Yaskawa INFORM job: DEMO_ROOF_UPPER_0625_3PAINT_38.JBI

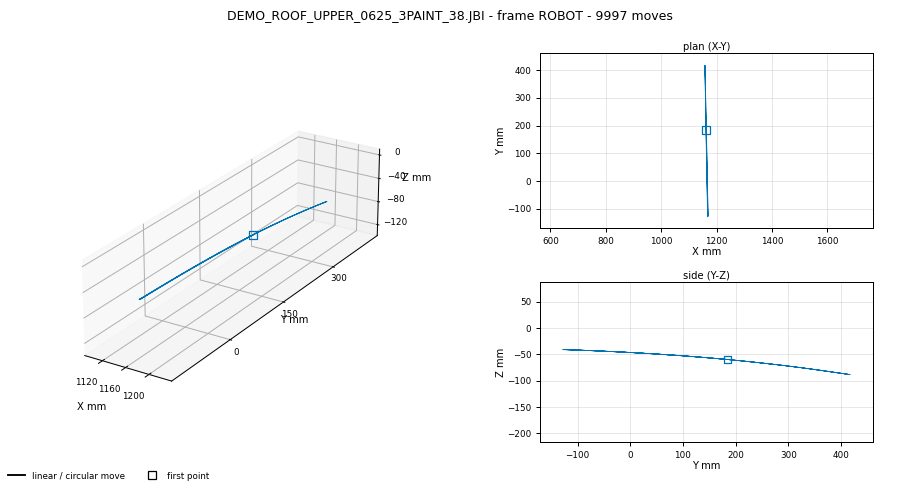
[picture p0: tool path of DEMO_ROOF_UPPER_0625_3PAINT_38.JBI in frame ROBOT, 9997 of 9997 moves have a stored position in this frame; points joined in program order, loops and branches not executed]
/JOB
//NAME DEMO_ROOF_UPPER_0625_3PAINT38
//POS
///NPOS 9997,0,0,0,0,0
///TOOL 0
///USER 0
///POSTYPE ROBOT
///RECTAN
///RCONF 1,0,0,0,0,0,0,0,0,0,0,0,0,0,0,0,0,0,0,0,0,0,0,0
C00000=1163.318,184.615,-59.683,-178.143,6.943,148.746
C00001=1163.323,184.345,-59.658,-178.145,6.942,148.747
C00002=1163.328,184.076,-59.633,-178.149,6.939,148.747
C00003=1163.333,183.807,-59.608,-178.152,6.936,148.747
C00004=1163.338,183.537,-59.582,-178.155,6.935,148.748
C00005=1163.342,183.288,-59.560,-178.157,6.933,148.748
C00006=1163.347,183.038,-59.537,-178.160,6.930,148.748
C00007=1163.352,182.789,-59.514,-178.163,6.928,148.748
C00008=1163.357,182.541,-59.491,-178.166,6.926,148.749
C00009=1163.361,182.292,-59.468,-178.169,6.924,148.749
C00010=1163.366,182.043,-59.445,-178.171,6.922,148.749
C00011=1163.370,181.794,-59.423,-178.174,6.920,148.750
C00012=1163.375,181.545,-59.399,-178.176,6.918,148.750
C00013=1163.379,181.297,-59.377,-178.180,6.916,148.750
C00014=1163.384,181.048,-59.353,-178.182,6.914,148.750
C00015=1163.389,180.799,-59.330,-178.185,6.912,148.751
C00016=1163.393,180.549,-59.308,-178.188,6.909,148.751
C00017=1163.398,180.300,-59.285,-178.190,6.907,148.752
C00018=1163.402,180.052,-59.262,-178.193,6.905,148.752
C00019=1163.407,179.803,-59.240,-178.195,6.904,148.752
C00020=1163.411,179.554,-59.217,-178.199,6.901,148.752
C00021=1163.416,179.305,-59.193,-178.201,6.899,148.753
C00022=1163.422,179.056,-59.171,-178.204,6.898,148.753
C00023=1163.426,178.807,-59.148,-178.206,6.895,148.753
C00024=1163.430,178.558,-59.125,-178.209,6.893,148.754
C00025=1163.435,178.309,-59.103,-178.212,6.891,148.754
C00026=1163.440,178.061,-59.080,-178.215,6.889,148.754
C00027=1163.444,177.811,-59.058,-178.217,6.887,148.754
C00028=1163.449,177.562,-59.035,-178.220,6.885,148.755
C00029=1163.453,177.314,-59.012,-178.223,6.883,148.755
C00030=1163.458,177.065,-58.990,-178.226,6.881,148.755
C00031=1163.462,176.816,-58.967,-178.228,6.879,148.756
C00032=1163.468,176.567,-58.945,-178.231,6.876,148.756
C00033=1163.472,176.318,-58.922,-178.234,6.875,148.756
C00034=1163.477,176.069,-58.899,-178.237,6.873,148.757
C00035=1163.482,175.821,-58.877,-178.239,6.871,148.757
C00036=1163.486,175.571,-58.855,-178.242,6.869,148.757
C00037=1163.491,175.322,-58.831,-178.245,6.867,148.758
C00038=1163.495,175.074,-58.810,-178.247,6.865,148.758
C00039=1163.500,174.824,-58.786,-178.250,6.863,148.758
C00040=1163.504,174.575,-58.764,-178.253,6.861,148.759
C00041=1163.510,174.327,-58.741,-178.256,6.859,148.759
C00042=1163.514,174.077,-58.719,-178.258,6.857,148.759
C00043=1163.518,173.829,-58.696,-178.261,6.855,148.760
C00044=1163.523,173.580,-58.674,-178.264,6.853,148.760
C00045=1163.528,173.330,-58.652,-178.267,6.851,148.760
C00046=1163.532,173.082,-58.629,-178.270,6.849,148.761
C00047=1163.537,172.833,-58.607,-178.272,6.847,148.761
C00048=1163.542,172.583,-58.585,-178.274,6.845,148.761
C00049=1163.547,172.335,-58.562,-178.277,6.843,148.761
C00050=1163.551,172.086,-58.540,-178.280,6.841,148.762
C00051=1163.555,171.836,-58.518,-178.283,6.839,148.762
C00052=1163.560,171.588,-58.496,-178.286,6.837,148.763
C00053=1163.565,171.339,-58.473,-178.289,6.835,148.763
C00054=1163.570,171.090,-58.451,-178.291,6.833,148.763
C00055=1163.574,170.841,-58.428,-178.294,6.831,148.763
C00056=1163.579,170.592,-58.406,-178.297,6.829,148.764
C00057=1163.584,170.343,-58.384,-178.299,6.827,148.764
C00058=1163.588,170.094,-58.362,-178.302,6.825,148.765
C00059=1163.593,169.845,-58.339,-178.305,6.824,148.765
C00060=1163.598,169.596,-58.317,-178.308,6.821,148.765
C00061=1163.602,169.347,-58.295,-178.310,6.819,148.765
C00062=1163.607,169.098,-58.273,-178.313,6.817,148.766
C00063=1163.612,168.849,-58.251,-178.316,6.815,148.766
C00064=1163.616,168.600,-58.228,-178.318,6.814,148.766
C00065=1163.621,168.352,-58.207,-178.322,6.811,148.767
C00066=1163.625,168.102,-58.185,-178.324,6.809,148.767
C00067=1163.630,167.854,-58.163,-178.326,6.807,148.767
C00068=1163.635,167.604,-58.140,-178.329,6.806,148.768
C00069=1163.640,167.356,-58.119,-178.332,6.804,148.768
C00070=1163.644,167.106,-58.096,-178.335,6.802,148.768
C00071=1163.649,166.858,-58.075,-178.338,6.800,148.769
C00072=1163.654,166.608,-58.053,-178.341,6.798,148.769
C00073=1163.658,166.360,-58.030,-178.343,6.796,148.770
C00074=1163.663,166.111,-58.008,-178.346,6.794,148.770
C00075=1163.668,165.862,-57.986,-178.348,6.792,148.770
C00076=1163.672,165.613,-57.964,-178.351,6.790,148.770
C00077=1163.677,165.364,-57.942,-178.354,6.788,148.771
C00078=1163.681,165.115,-57.920,-178.357,6.786,148.771
C00079=1163.686,164.866,-57.899,-178.359,6.784,148.772
C00080=1163.691,164.617,-57.877,-178.362,6.783,148.772
C00081=1163.695,164.368,-57.855,-178.365,6.781,148.772
C00082=1163.700,164.119,-57.833,-178.368,6.779,148.773
C00083=1163.705,163.870,-57.811,-178.370,6.777,148.773
C00084=1163.710,163.621,-57.789,-178.373,6.774,148.773
C00085=1163.715,163.371,-57.767,-178.376,6.773,148.774
C00086=1163.720,163.122,-57.746,-178.378,6.771,148.774
C00087=1163.724,162.873,-57.724,-178.381,6.769,148.774
C00088=1163.729,162.624,-57.702,-178.384,6.767,148.775
C00089=1163.734,162.376,-57.680,-178.386,6.766,148.775
C00090=1163.738,162.126,-57.658,-178.389,6.764,148.775
C00091=1163.743,161.878,-57.637,-178.392,6.761,148.776
C00092=1163.747,161.628,-57.615,-178.395,6.760,148.776
C00093=1163.752,161.379,-57.594,-178.397,6.758,148.776
C00094=1163.757,161.131,-57.572,-178.400,6.756,148.777
C00095=1163.761,160.881,-57.550,-178.403,6.754,148.777
C00096=1163.766,160.633,-57.528,-178.405,6.752,148.777
C00097=1163.770,160.383,-57.506,-178.408,6.751,148.778
C00098=1163.775,160.135,-57.485,-178.411,6.749,148.778
C00099=1163.780,159.885,-57.464,-178.414,6.746,148.778
C00100=1163.785,159.636,-57.441,-178.417,6.745,148.779
C00101=1163.790,159.387,-57.420,-178.419,6.743,148.779
C00102=1163.794,159.139,-57.399,-178.422,6.741,148.780
C00103=1163.798,158.889,-57.377,-178.425,6.739,148.780
C00104=1163.803,158.640,-57.356,-178.428,6.738,148.780
C00105=1163.809,158.371,-57.332,-178.430,6.736,148.781
C00106=1163.813,158.103,-57.309,-178.434,6.733,148.781
C00107=1163.819,157.833,-57.286,-178.436,6.731,148.781
C00108=1163.823,157.564,-57.263,-178.440,6.729,148.782
C00109=1163.828,157.316,-57.241,-178.442,6.727,148.782
C00110=1163.833,157.066,-57.220,-178.445,6.725,148.783
C00111=1163.838,156.817,-57.198,-178.448,6.724,148.783
C00112=1163.843,156.568,-57.176,-178.450,6.722,148.783
C00113=1163.848,156.319,-57.155,-178.453,6.720,148.784
C00114=1163.852,156.071,-57.134,-178.456,6.718,148.784
C00115=1163.856,155.821,-57.113,-178.458,6.717,148.784
C00116=1163.861,155.572,-57.091,-178.461,6.715,148.785
C00117=1163.866,155.324,-57.070,-178.464,6.713,148.785
C00118=1163.871,155.074,-57.048,-178.466,6.711,148.785
C00119=1163.876,154.825,-57.027,-178.469,6.709,148.786
C00120=1163.880,154.576,-57.006,-178.472,6.707,148.786
C00121=1163.885,154.327,-56.985,-178.475,6.705,148.786
C00122=1163.889,154.077,-56.963,-178.477,6.703,148.787
C00123=1163.894,153.829,-56.942,-178.480,6.702,148.787
C00124=1163.899,153.580,-56.921,-178.483,6.700,148.788
C00125=1163.904,153.331,-56.899,-178.485,6.698,148.788
C00126=1163.909,153.082,-56.879,-178.488,6.696,148.788
C00127=1163.913,152.833,-56.856,-178.491,6.695,148.789
C00128=1163.918,152.584,-56.836,-178.494,6.693,148.789
C00129=1163.923,152.334,-56.815,-178.496,6.691,148.790
C00130=1163.928,152.086,-56.793,-178.499,6.689,148.790
C00131=1163.932,151.836,-56.772,-178.502,6.688,148.790
C00132=1163.936,151.587,-56.751,-178.504,6.686,148.791
C00133=1163.941,151.338,-56.730,-178.507,6.684,148.791
C00134=1163.947,151.089,-56.709,-178.510,6.682,148.791
C00135=1163.951,150.841,-56.688,-178.513,6.680,148.792
C00136=1163.956,150.591,-56.667,-178.516,6.678,148.792
C00137=1163.960,150.341,-56.646,-178.518,6.676,148.793
C00138=1163.965,150.093,-56.625,-178.521,6.675,148.793
C00139=1163.970,149.844,-56.604,-178.524,6.673,148.793
C00140=1163.975,149.594,-56.583,-178.527,6.671,148.794
C00141=1163.979,149.346,-56.562,-178.529,6.669,148.794
C00142=1163.984,149.097,-56.541,-178.532,6.668,148.794
C00143=1163.989,148.848,-56.520,-178.535,6.666,148.795
C00144=1163.993,148.598,-56.499,-178.537,6.664,148.795
C00145=1163.998,148.349,-56.477,-178.540,6.663,148.796
C00146=1164.003,148.100,-56.457,-178.543,6.661,148.796
C00147=1164.008,147.851,-56.436,-178.545,6.659,148.796
C00148=1164.013,147.602,-56.415,-178.548,6.657,148.797
C00149=1164.017,147.354,-56.394,-178.551,6.656,148.797
C00150=1164.022,147.104,-56.373,-178.554,6.654,148.798
C00151=1164.027,146.855,-56.353,-178.556,6.652,148.798
C00152=1164.031,146.605,-56.331,-178.559,6.650,148.798
C00153=1164.036,146.356,-56.311,-178.562,6.649,148.799
C00154=1164.041,146.107,-56.290,-178.564,6.647,148.799
C00155=1164.045,145.859,-56.269,-178.567,6.645,148.799
C00156=1164.050,145.610,-56.248,-178.570,6.643,148.800
C00157=1164.055,145.361,-56.227,-178.572,6.642,148.800
C00158=1164.060,145.111,-56.206,-178.575,6.640,148.801
C00159=1164.064,144.862,-56.186,-178.578,6.638,148.801
C00160=1164.069,144.613,-56.165,-178.581,6.636,148.801
C00161=1164.074,144.364,-56.145,-178.583,6.635,148.802
C00162=1164.079,144.115,-56.124,-178.586,6.633,148.802
C00163=1164.083,143.866,-56.103,-178.589,6.631,148.803
C00164=1164.089,143.617,-56.082,-178.591,6.630,148.803
C00165=1164.093,143.368,-56.062,-178.594,6.628,148.803
C00166=1164.098,143.118,-56.041,-178.597,6.626,148.804
C00167=1164.102,142.869,-56.020,-178.600,6.625,148.804
C00168=1164.107,142.620,-56.000,-178.603,6.623,148.805
C00169=1164.112,142.371,-55.979,-178.605,6.621,148.805
C00170=1164.116,142.122,-55.959,-178.608,6.619,148.805
C00171=1164.121,141.872,-55.938,-178.611,6.618,148.806
C00172=1164.126,141.624,-55.917,-178.613,6.616,148.806
C00173=1164.130,141.375,-55.897,-178.616,6.614,148.807
C00174=1164.135,141.125,-55.876,-178.619,6.613,148.807
C00175=1164.140,140.876,-55.856,-178.622,6.611,148.807
C00176=1164.145,140.627,-55.835,-178.624,6.609,148.808
C00177=1164.149,140.378,-55.814,-178.627,6.607,148.808
C00178=1164.154,140.129,-55.794,-178.630,6.606,148.809
C00179=1164.159,139.880,-55.773,-178.632,6.604,148.809
C00180=1164.164,139.630,-55.753,-178.635,6.602,148.809
C00181=1164.169,139.382,-55.733,-178.638,6.600,148.810
C00182=1164.174,139.133,-55.712,-178.640,6.599,148.810
C00183=1164.178,138.884,-55.692,-178.643,6.597,148.810
C00184=1164.183,138.635,-55.672,-178.646,6.596,148.811
C00185=1164.188,138.386,-55.651,-178.649,6.594,148.811
C00186=1164.193,138.136,-55.631,-178.652,6.592,148.812
C00187=1164.197,137.887,-55.611,-178.654,6.590,148.812
C00188=1164.202,137.638,-55.590,-178.657,6.589,148.813
C00189=1164.207,137.389,-55.569,-178.660,6.587,148.813
C00190=1164.212,137.139,-55.550,-178.663,6.585,148.813
C00191=1164.216,136.890,-55.529,-178.665,6.583,148.814
C00192=1164.220,136.642,-55.509,-178.668,6.582,148.814
C00193=1164.226,136.392,-55.488,-178.671,6.580,148.815
C00194=1164.230,136.143,-55.468,-178.673,6.579,148.815
C00195=1164.235,135.894,-55.448,-178.676,6.577,148.815
C00196=1164.240,135.646,-55.428,-178.679,6.576,148.816
C00197=1164.245,135.396,-55.408,-178.681,6.574,148.816
C00198=1164.250,135.147,-55.387,-178.684,6.572,148.817
C00199=1164.254,134.898,-55.367,-178.687,6.571,148.817
C00200=1164.259,134.648,-55.347,-178.690,6.569,148.818
C00201=1164.263,134.399,-55.327,-178.692,6.567,148.818
C00202=1164.269,134.150,-55.306,-178.695,6.566,148.818
C00203=1164.274,133.901,-55.287,-178.698,6.564,148.819
C00204=1164.278,133.652,-55.266,-178.700,6.562,148.819
C00205=1164.283,133.403,-55.247,-178.703,6.560,148.820
C00206=1164.287,133.154,-55.226,-178.706,6.559,148.820
C00207=1164.292,132.905,-55.206,-178.709,6.557,148.821
C00208=1164.297,132.655,-55.186,-178.712,6.556,148.821
C00209=1164.302,132.386,-55.164,-178.714,6.554,148.821
C00210=1164.307,132.118,-55.143,-178.717,6.552,148.822
C00211=1164.313,131.849,-55.121,-178.720,6.551,148.822
C00212=1164.318,131.580,-55.100,-178.723,6.549,148.823
C00213=1164.323,131.332,-55.080,-178.726,6.547,148.823
C00214=1164.327,131.083,-55.060,-178.728,6.546,148.823
C00215=1164.332,130.833,-55.039,-178.731,6.544,148.824
C00216=1164.337,130.584,-55.020,-178.734,6.542,148.824
C00217=1164.342,130.335,-54.999,-178.737,6.540,148.825
C00218=1164.347,130.086,-54.980,-178.740,6.539,148.825
C00219=1164.351,129.837,-54.960,-178.742,6.538,148.826
C00220=1164.356,129.588,-54.940,-178.745,6.536,148.826
C00221=1164.361,129.339,-54.920,-178.747,6.535,148.826
C00222=1164.366,129.090,-54.900,-178.750,6.533,148.827
C00223=1164.371,128.840,-54.881,-178.753,6.531,148.827
C00224=1164.375,128.591,-54.860,-178.755,6.529,148.828
C00225=1164.380,128.342,-54.841,-178.758,6.528,148.828
C00226=1164.385,128.093,-54.821,-178.761,6.526,148.829
C00227=1164.390,127.844,-54.801,-178.764,6.525,148.829
C00228=1164.394,127.594,-54.781,-178.766,6.524,148.829
C00229=1164.399,127.345,-54.762,-178.769,6.522,148.830
C00230=1164.404,127.096,-54.742,-178.772,6.520,148.830
C00231=1164.409,126.847,-54.722,-178.774,6.519,148.831
C00232=1164.414,126.597,-54.702,-178.777,6.517,148.831
C00233=1164.418,126.348,-54.682,-178.780,6.515,148.832
C00234=1164.423,126.099,-54.663,-178.783,6.514,148.832
C00235=1164.428,125.850,-54.643,-178.786,6.512,148.832
C00236=1164.432,125.601,-54.624,-178.788,6.510,148.833
C00237=1164.437,125.352,-54.604,-178.790,6.509,148.833
C00238=1164.442,125.103,-54.584,-178.793,6.508,148.834
C00239=1164.447,124.853,-54.565,-178.796,6.506,148.834
C00240=1164.452,124.604,-54.545,-178.799,6.505,148.835
C00241=1164.456,124.355,-54.525,-178.802,6.503,148.835
C00242=1164.461,124.106,-54.505,-178.804,6.501,148.835
C00243=1164.467,123.857,-54.486,-178.807,6.499,148.836
C00244=1164.471,123.607,-54.466,-178.809,6.498,148.836
C00245=1164.475,123.358,-54.447,-178.812,6.497,148.837
C00246=1164.481,123.109,-54.428,-178.815,6.495,148.837
C00247=1164.485,122.860,-54.408,-178.818,6.494,148.838
C00248=1164.490,122.611,-54.388,-178.821,6.492,148.838
C00249=1164.495,122.362,-54.369,-178.823,6.490,148.838
C00250=1164.500,122.112,-54.349,-178.826,6.489,148.839
C00251=1164.504,121.863,-54.330,-178.829,6.488,148.840
C00252=1164.509,121.614,-54.311,-178.831,6.486,148.840
C00253=1164.514,121.365,-54.291,-178.834,6.485,148.840
C00254=1164.519,121.116,-54.272,-178.837,6.483,148.841
C00255=1164.524,120.866,-54.252,-178.839,6.481,148.841
C00256=1164.528,120.617,-54.233,-178.842,6.479,148.842
C00257=1164.533,120.368,-54.214,-178.845,6.479,148.842
C00258=1164.538,120.119,-54.194,-178.847,6.477,148.843
C00259=1164.544,119.870,-54.175,-178.850,6.475,148.843
C00260=1164.548,119.620,-54.156,-178.853,6.474,148.843
C00261=1164.552,119.371,-54.136,-178.856,6.472,148.844
C00262=1164.558,119.122,-54.117,-178.859,6.471,148.844
C00263=1164.562,118.872,-54.097,-178.861,6.470,148.845
C00264=1164.567,118.624,-54.078,-178.864,6.468,148.845
C00265=1164.572,118.374,-54.059,-178.866,6.466,148.846
C00266=1164.577,118.125,-54.039,-178.869,6.464,148.846
C00267=1164.581,117.876,-54.020,-178.872,6.463,148.847
C00268=1164.586,117.627,-54.001,-178.874,6.462,148.847
C00269=1164.591,117.378,-53.981,-178.877,6.461,148.847
C00270=1164.595,117.128,-53.962,-178.880,6.459,148.848
C00271=1164.601,116.880,-53.943,-178.883,6.457,148.848
C00272=1164.606,116.629,-53.924,-178.886,6.456,148.849
C00273=1164.610,116.381,-53.905,-178.888,6.455,148.849
C00274=1164.615,116.131,-53.886,-178.891,6.453,148.850
C00275=1164.620,115.882,-53.866,-178.893,6.451,148.850
C00276=1164.624,115.633,-53.847,-178.896,6.450,148.850
C00277=1164.630,115.384,-53.828,-178.899,6.448,148.851
C00278=1164.635,115.134,-53.809,-178.901,6.447,148.852
C00279=1164.639,114.886,-53.790,-178.904,6.446,148.852
C00280=1164.644,114.636,-53.771,-178.907,6.444,148.852
C00281=1164.649,114.387,-53.752,-178.910,6.443,148.853
C00282=1164.654,114.137,-53.733,-178.913,6.441,148.853
C00283=1164.659,113.888,-53.714,-178.915,6.440,148.854
C00284=1164.663,113.639,-53.695,-178.918,6.438,148.854
C00285=1164.668,113.390,-53.676,-178.920,6.437,148.855
C00286=1164.673,113.140,-53.657,-178.923,6.435,148.855
C00287=1164.678,112.891,-53.638,-178.926,6.433,148.856
C00288=1164.682,112.642,-53.619,-178.928,6.433,148.856
C00289=1164.688,112.393,-53.600,-178.931,6.431,148.856
C00290=1164.693,112.144,-53.581,-178.934,6.430,148.857
C00291=1164.697,111.895,-53.562,-178.937,6.428,148.857
C00292=1164.703,111.645,-53.543,-178.939,6.427,148.858
C00293=1164.707,111.396,-53.524,-178.942,6.425,148.858
C00294=1164.712,111.147,-53.505,-178.945,6.424,148.859
C00295=1164.716,110.897,-53.487,-178.948,6.422,148.859
C00296=1164.722,110.648,-53.467,-178.950,6.420,148.860
C00297=1164.726,110.400,-53.449,-178.953,6.419,148.860
C00298=1164.731,110.150,-53.430,-178.955,6.418,148.861
C00299=1164.736,109.901,-53.411,-178.958,6.416,148.861
C00300=1164.741,109.651,-53.392,-178.961,6.415,148.862
C00301=1164.746,109.402,-53.373,-178.963,6.414,148.862
C00302=1164.750,109.153,-53.355,-178.966,6.412,148.862
C00303=1164.755,108.903,-53.336,-178.969,6.411,148.863
C00304=1164.760,108.655,-53.317,-178.972,6.409,148.863
C00305=1164.765,108.405,-53.298,-178.974,6.408,148.864
C00306=1164.770,108.156,-53.279,-178.977,6.406,148.864
C00307=1164.775,107.907,-53.261,-178.980,6.405,148.865
C00308=1164.779,107.657,-53.242,-178.983,6.403,148.865
C00309=1164.784,107.408,-53.224,-178.985,6.402,148.866
C00310=1164.789,107.159,-53.204,-178.988,6.401,148.866
C00311=1164.794,106.910,-53.186,-178.991,6.399,148.867
C00312=1164.799,106.660,-53.168,-178.993,6.398,148.867
C00313=1164.804,106.392,-53.147,-178.996,6.397,148.868
C00314=1164.809,106.123,-53.127,-178.999,6.395,148.868
C00315=1164.814,105.855,-53.108,-179.002,6.394,148.869
C00316=1164.820,105.587,-53.087,-179.005,6.392,148.869
C00317=1164.825,105.338,-53.069,-179.007,6.391,148.870
C00318=1164.829,105.089,-53.050,-179.010,6.389,148.870
C00319=1164.835,104.839,-53.031,-179.013,6.388,148.871
C00320=1164.839,104.590,-53.013,-179.016,6.387,148.871
C00321=1164.843,104.341,-52.994,-179.018,6.385,148.872
C00322=1164.848,104.091,-52.976,-179.021,6.383,148.872
C00323=1164.854,103.842,-52.958,-179.024,6.383,148.873
C00324=1164.858,103.593,-52.939,-179.026,6.381,148.873
C00325=1164.863,103.343,-52.921,-179.029,6.379,148.873
C00326=1164.869,103.094,-52.902,-179.032,6.378,148.874
C00327=1164.873,102.845,-52.883,-179.034,6.377,148.874
C00328=1164.877,102.596,-52.865,-179.037,6.375,148.875
C00329=1164.882,102.346,-52.847,-179.040,6.374,148.875
C00330=1164.888,102.097,-52.829,-179.042,6.373,148.876
C00331=1164.893,101.848,-52.810,-179.045,6.371,148.876
C00332=1164.897,101.598,-52.791,-179.048,6.370,148.877
C00333=1164.902,101.349,-52.774,-179.050,6.369,148.877
C00334=1164.908,101.100,-52.755,-179.053,6.367,148.878
C00335=1164.912,100.851,-52.737,-179.056,6.366,148.878
C00336=1164.916,100.601,-52.718,-179.059,6.364,148.879
C00337=1164.921,100.352,-52.700,-179.061,6.364,148.879
C00338=1164.926,100.103,-52.682,-179.064,6.362,148.880
C00339=1164.932,99.854,-52.663,-179.067,6.360,148.880
C00340=1164.936,99.604,-52.645,-179.069,6.360,148.881
C00341=1164.941,99.355,-52.626,-179.072,6.358,148.881
C00342=1164.946,99.106,-52.608,-179.075,6.356,148.882
C00343=1164.951,98.857,-52.590,-179.077,6.356,148.882
C00344=1164.956,98.608,-52.572,-179.080,6.354,148.883
C00345=1164.960,98.358,-52.554,-179.083,6.352,148.883
C00346=1164.966,98.108,-52.535,-179.085,6.351,148.883
C00347=1164.970,97.859,-52.517,-179.088,6.350,148.884
C00348=1164.975,97.610,-52.499,-179.091,6.348,148.885
C00349=1164.980,97.361,-52.482,-179.093,6.347,148.885
C00350=1164.985,97.112,-52.464,-179.096,6.346,148.886
C00351=1164.990,96.862,-52.445,-179.099,6.344,148.886
C00352=1164.994,96.612,-52.427,-179.101,6.343,148.886
C00353=1164.999,96.363,-52.409,-179.104,6.342,148.887
C00354=1165.004,96.114,-52.391,-179.107,6.340,148.887
C00355=1165.010,95.865,-52.373,-179.109,6.340,148.888
C00356=1165.015,95.615,-52.355,-179.112,6.338,148.889
C00357=1165.019,95.366,-52.336,-179.115,6.336,148.889
C00358=1165.024,95.116,-52.318,-179.117,6.336,148.889
C00359=1165.029,94.867,-52.300,-179.120,6.334,148.890
C00360=1165.034,94.618,-52.282,-179.123,6.333,148.890
C00361=1165.039,94.369,-52.264,-179.125,6.332,148.891
C00362=1165.044,94.120,-52.246,-179.129,6.330,148.892
C00363=1165.049,93.871,-52.228,-179.131,6.329,148.892
C00364=1165.053,93.621,-52.210,-179.133,6.328,148.892
C00365=1165.058,93.372,-52.193,-179.137,6.326,148.893
C00366=1165.063,93.122,-52.174,-179.139,6.325,148.893
C00367=1165.068,92.873,-52.156,-179.141,6.324,148.894
C00368=1165.073,92.624,-52.138,-179.145,6.322,148.894
C00369=1165.077,92.375,-52.120,-179.147,6.321,148.895
C00370=1165.083,92.125,-52.103,-179.150,6.320,148.895
C00371=1165.088,91.876,-52.085,-179.153,6.319,148.896
C00372=1165.092,91.627,-52.067,-179.155,6.318,148.896
C00373=1165.097,91.377,-52.049,-179.158,6.316,148.897
C00374=1165.102,91.128,-52.031,-179.161,6.315,148.897
C00375=1165.107,90.879,-52.014,-179.163,6.314,148.898
C00376=1165.112,90.630,-51.996,-179.166,6.312,148.898
C00377=1165.117,90.380,-51.978,-179.169,6.311,148.899
C00378=1165.122,90.131,-51.960,-179.171,6.310,148.899
C00379=1165.126,89.882,-51.942,-179.174,6.308,148.900
C00380=1165.132,89.632,-51.925,-179.176,6.308,148.900
C00381=1165.137,89.383,-51.907,-179.179,6.306,148.901
C00382=1165.141,89.133,-51.889,-179.182,6.304,148.901
C00383=1165.146,88.884,-51.871,-179.184,6.304,148.902
C00384=1165.151,88.634,-51.854,-179.187,6.302,148.902
C00385=1165.155,88.385,-51.836,-179.190,6.300,148.903
C00386=1165.160,88.136,-51.818,-179.193,6.300,148.903
C00387=1165.165,87.886,-51.801,-179.195,6.298,148.904
C00388=1165.170,87.637,-51.783,-179.197,6.297,148.904
C00389=1165.175,87.388,-51.765,-179.201,6.296,148.905
C00390=1165.180,87.138,-51.748,-179.203,6.294,148.905
C00391=1165.185,86.889,-51.730,-179.206,6.294,148.906
C00392=1165.189,86.640,-51.712,-179.209,6.292,148.906
C00393=1165.195,86.391,-51.696,-179.211,6.291,148.907
C00394=1165.200,86.142,-51.678,-179.214,6.290,148.907
C00395=1165.205,85.892,-51.660,-179.217,6.288,148.908
C00396=1165.210,85.643,-51.643,-179.219,6.287,148.908
C00397=1165.214,85.394,-51.625,-179.222,6.286,148.909
C00398=1165.220,85.144,-51.608,-179.224,6.285,148.909
C00399=1165.225,84.895,-51.590,-179.227,6.283,148.910
C00400=1165.229,84.646,-51.573,-179.230,6.283,148.910
C00401=1165.234,84.397,-51.555,-179.232,6.281,148.911
C00402=1165.239,84.147,-51.538,-179.236,6.280,148.912
C00403=1165.244,83.898,-51.520,-179.238,6.279,148.912
C00404=1165.249,83.648,-51.503,-179.240,6.277,148.912
C00405=1165.254,83.399,-51.485,-179.243,6.277,148.913
C00406=1165.259,83.149,-51.468,-179.246,6.275,148.913
C00407=1165.264,82.900,-51.450,-179.249,6.273,148.914
C00408=1165.268,82.650,-51.433,-179.251,6.273,148.915
C00409=1165.273,82.401,-51.415,-179.254,6.271,148.915
C00410=1165.279,82.152,-51.398,-179.256,6.270,148.916
C00411=1165.283,81.903,-51.381,-179.259,6.269,148.916
C00412=1165.288,81.653,-51.364,-179.261,6.268,148.916
C00413=1165.293,81.404,-51.346,-179.265,6.266,148.917
C00414=1165.298,81.155,-51.329,-179.267,6.265,148.918
C00415=1165.303,80.905,-51.312,-179.270,6.264,148.918
C00416=1165.308,80.656,-51.294,-179.273,6.263,148.919
C00417=1165.313,80.388,-51.276,-179.275,6.262,148.919
C00418=1165.318,80.119,-51.257,-179.278,6.260,148.920
C00419=1165.324,79.851,-51.238,-179.281,6.259,148.920
C00420=1165.329,79.583,-51.220,-179.284,6.257,148.921
C00421=1165.334,79.333,-51.203,-179.287,6.257,148.921
C00422=1165.339,79.083,-51.186,-179.289,6.255,148.922
C00423=1165.343,78.835,-51.168,-179.291,6.254,148.922
C00424=1165.349,78.585,-51.151,-179.295,6.253,148.923
C00425=1165.354,78.335,-51.134,-179.297,6.252,148.923
C00426=1165.359,78.087,-51.117,-179.300,6.251,148.924
C00427=1165.364,77.837,-51.099,-179.302,6.250,148.924
C00428=1165.368,77.588,-51.083,-179.305,6.248,148.925
C00429=1165.373,77.338,-51.065,-179.308,6.247,148.925
C00430=1165.378,77.089,-51.048,-179.310,6.246,148.926
C00431=1165.383,76.839,-51.031,-179.313,6.245,148.927
C00432=1165.388,76.590,-51.015,-179.316,6.244,148.927
C00433=1165.393,76.340,-50.997,-179.318,6.242,148.927
C00434=1165.397,76.092,-50.980,-179.321,6.242,148.928
C00435=1165.403,75.842,-50.963,-179.324,6.240,148.929
C00436=1165.408,75.593,-50.946,-179.326,6.239,148.929
C00437=1165.413,75.343,-50.929,-179.329,6.238,148.930
C00438=1165.418,75.093,-50.912,-179.331,6.237,148.930
C00439=1165.422,74.845,-50.894,-179.334,6.235,148.931
C00440=1165.427,74.595,-50.878,-179.337,6.235,148.931
C00441=1165.433,74.346,-50.861,-179.340,6.233,148.932
C00442=1165.437,74.097,-50.844,-179.342,6.232,148.932
C00443=1165.442,73.847,-50.827,-179.345,6.231,148.933
C00444=1165.447,73.597,-50.810,-179.347,6.230,148.933
C00445=1165.453,73.348,-50.793,-179.350,6.228,148.934
C00446=1165.457,73.099,-50.776,-179.353,6.228,148.934
C00447=1165.462,72.849,-50.759,-179.355,6.226,148.935
C00448=1165.466,72.600,-50.742,-179.358,6.226,148.935
C00449=1165.472,72.351,-50.725,-179.361,6.224,148.936
C00450=1165.477,72.101,-50.709,-179.363,6.223,148.936
C00451=1165.481,71.852,-50.692,-179.366,6.222,148.937
C00452=1165.487,71.603,-50.675,-179.368,6.221,148.937
C00453=1165.492,71.353,-50.658,-179.372,6.220,148.938
C00454=1165.497,71.104,-50.641,-179.374,6.219,148.939
C00455=1165.501,70.854,-50.624,-179.377,6.217,148.939
C00456=1165.506,70.605,-50.608,-179.379,6.217,148.940
C00457=1165.512,70.356,-50.591,-179.382,6.215,148.940
C00458=1165.516,70.106,-50.574,-179.384,6.214,148.941
C00459=1165.521,69.857,-50.558,-179.387,6.213,148.941
C00460=1165.526,69.607,-50.541,-179.390,6.212,148.942
C00461=1165.531,69.358,-50.524,-179.393,6.211,148.942
C00462=1165.536,69.109,-50.508,-179.395,6.210,148.943
C00463=1165.541,68.859,-50.490,-179.398,6.208,148.943
C00464=1165.546,68.610,-50.474,-179.400,6.208,148.944
C00465=1165.551,68.361,-50.457,-179.403,6.206,148.944
C00466=1165.556,68.111,-50.441,-179.405,6.205,148.945
C00467=1165.561,67.861,-50.424,-179.409,6.204,148.945
C00468=1165.566,67.612,-50.408,-179.411,6.203,148.946
C00469=1165.571,67.363,-50.391,-179.414,6.202,148.947
C00470=1165.575,67.113,-50.374,-179.416,6.201,148.947
C00471=1165.580,66.864,-50.358,-179.419,6.200,148.948
C00472=1165.585,66.615,-50.341,-179.421,6.199,148.948
C00473=1165.591,66.366,-50.324,-179.424,6.198,148.949
C00474=1165.596,66.116,-50.308,-179.427,6.197,148.949
C00475=1165.600,65.866,-50.291,-179.429,6.196,148.950
C00476=1165.605,65.617,-50.275,-179.432,6.194,148.950
C00477=1165.610,65.368,-50.258,-179.434,6.193,148.951
C00478=1165.615,65.119,-50.242,-179.438,6.192,148.951
C00479=1165.620,64.869,-50.226,-179.440,6.191,148.952
C00480=1165.625,64.619,-50.209,-179.443,6.190,148.952
C00481=1165.630,64.370,-50.193,-179.445,6.189,148.953
C00482=1165.635,64.121,-50.175,-179.448,6.188,148.954
C00483=1165.640,63.871,-50.160,-179.450,6.187,148.954
C00484=1165.645,63.622,-50.143,-179.453,6.186,148.954
C00485=1165.649,63.372,-50.126,-179.456,6.185,148.955
C00486=1165.654,63.124,-50.110,-179.458,6.184,148.956
C00487=1165.660,62.873,-50.094,-179.461,6.183,148.956
C00488=1165.665,62.624,-50.077,-179.463,6.182,148.957
C00489=1165.670,62.375,-50.061,-179.467,6.180,148.957
C00490=1165.675,62.125,-50.045,-179.469,6.179,148.958
C00491=1165.679,61.876,-50.028,-179.472,6.178,148.958
C00492=1165.684,61.627,-50.012,-179.474,6.177,148.959
C00493=1165.689,61.377,-49.996,-179.477,6.177,148.959
C00494=1165.694,61.127,-49.979,-179.480,6.175,148.960
C00495=1165.700,60.879,-49.962,-179.482,6.175,148.961
C00496=1165.704,60.628,-49.947,-179.485,6.173,148.961
C00497=1165.709,60.380,-49.930,-179.487,6.172,148.961
C00498=1165.714,60.130,-49.914,-179.490,6.171,148.962
C00499=1165.719,59.881,-49.898,-179.492,6.170,148.963
C00500=1165.724,59.631,-49.881,-179.495,6.169,148.963
C00501=1165.729,59.382,-49.866,-179.498,6.168,148.964
C00502=1165.734,59.132,-49.849,-179.500,6.167,148.964
C00503=1165.739,58.883,-49.833,-179.503,6.166,148.965
C00504=1165.743,58.633,-49.817,-179.506,6.165,148.965
C00505=1165.750,58.384,-49.801,-179.508,6.164,148.966
C00506=1165.754,58.134,-49.784,-179.511,6.163,148.967
C00507=1165.759,57.885,-49.768,-179.513,6.162,148.967
C00508=1165.765,57.636,-49.752,-179.517,6.161,148.968
C00509=1165.769,57.386,-49.736,-179.519,6.160,148.968
C00510=1165.774,57.137,-49.720,-179.522,6.158,148.969
C00511=1165.779,56.887,-49.704,-179.524,6.158,148.969
C00512=1165.784,56.638,-49.688,-179.527,6.157,148.970
C00513=1165.789,56.388,-49.672,-179.529,6.155,148.970
C00514=1165.794,56.139,-49.655,-179.532,6.155,148.971
C00515=1165.799,55.889,-49.639,-179.535,6.153,148.971
C00516=1165.804,55.641,-49.623,-179.537,6.153,148.972
C00517=1165.809,55.391,-49.607,-179.540,6.152,148.972
C00518=1165.814,55.141,-49.591,-179.542,6.150,148.973
C00519=1165.819,54.892,-49.575,-179.545,6.150,148.974
C00520=1165.824,54.642,-49.559,-179.547,6.149,148.974
C00521=1165.830,54.374,-49.542,-179.550,6.148,148.975
C00522=1165.835,54.105,-49.525,-179.554,6.146,148.975
C00523=1165.840,53.837,-49.507,-179.556,6.145,148.976
C00524=1165.845,53.568,-49.490,-179.559,6.144,148.976
C00525=1165.850,53.319,-49.475,-179.562,6.144,148.977
C00526=1165.855,53.070,-49.459,-179.564,6.143,148.978
C00527=1165.860,52.820,-49.443,-179.567,6.141,148.978
C00528=1165.865,52.571,-49.427,-179.569,6.141,148.979
C00529=1165.870,52.321,-49.411,-179.572,6.139,148.979
C00530=1165.875,52.072,-49.395,-179.575,6.138,148.980
C00531=1165.881,51.822,-49.379,-179.577,6.138,148.980
C00532=1165.885,51.572,-49.363,-179.580,6.136,148.981
C00533=1165.891,51.323,-49.348,-179.583,6.136,148.982
C00534=1165.895,51.075,-49.332,-179.585,6.135,148.982
C00535=1165.900,50.824,-49.316,-179.588,6.134,148.983
C00536=1165.905,50.575,-49.301,-179.590,6.133,148.983
C00537=1165.911,50.326,-49.285,-179.593,6.131,148.984
C00538=1165.915,50.076,-49.268,-179.595,6.131,148.984
C00539=1165.920,49.827,-49.253,-179.598,6.130,148.985
C00540=1165.925,49.577,-49.237,-179.601,6.128,148.985
C00541=1165.930,49.328,-49.222,-179.603,6.128,148.986
C00542=1165.935,49.078,-49.206,-179.606,6.127,148.986
C00543=1165.940,48.829,-49.190,-179.609,6.126,148.987
C00544=1165.945,48.579,-49.174,-179.611,6.125,148.988
C00545=1165.950,48.330,-49.159,-179.614,6.124,148.988
C00546=1165.955,48.081,-49.143,-179.616,6.123,148.989
C00547=1165.960,47.831,-49.127,-179.619,6.122,148.989
C00548=1165.965,47.581,-49.112,-179.621,6.121,148.990
C00549=1165.970,47.332,-49.097,-179.624,6.120,148.990
C00550=1165.975,47.082,-49.081,-179.627,6.119,148.991
C00551=1165.980,46.833,-49.065,-179.629,6.119,148.992
C00552=1165.985,46.584,-49.049,-179.632,6.117,148.992
C00553=1165.990,46.335,-49.034,-179.635,6.117,148.993
C00554=1165.995,46.085,-49.018,-179.637,6.116,148.993
C00555=1166.000,45.835,-49.002,-179.640,6.114,148.994
C00556=1166.006,45.586,-48.987,-179.642,6.113,148.994
C00557=1166.010,45.336,-48.972,-179.645,6.113,148.995
C00558=1166.015,45.087,-48.956,-179.648,6.111,148.995
C00559=1166.020,44.837,-48.940,-179.650,6.111,148.996
C00560=1166.025,44.588,-48.925,-179.652,6.110,148.996
C00561=1166.030,44.338,-48.909,-179.656,6.109,148.997
C00562=1166.035,44.089,-48.894,-179.658,6.108,148.998
C00563=1166.040,43.840,-48.879,-179.660,6.107,148.998
C00564=1166.045,43.590,-48.863,-179.663,6.106,148.999
C00565=1166.051,43.341,-48.848,-179.666,6.105,148.999
C00566=1166.055,43.091,-48.832,-179.668,6.104,149.000
C00567=1166.060,42.842,-48.817,-179.671,6.103,149.000
C00568=1166.065,42.592,-48.801,-179.673,6.102,149.001
C00569=1166.070,42.343,-48.786,-179.676,6.102,149.002
C00570=1166.075,42.093,-48.770,-179.679,6.100,149.002
C00571=1166.080,41.844,-48.755,-179.681,6.100,149.003
C00572=1166.085,41.594,-48.740,-179.684,6.099,149.003
C00573=1166.091,41.344,-48.725,-179.686,6.098,149.004
C00574=1166.095,41.095,-48.710,-179.689,6.097,149.005
C00575=1166.101,40.846,-48.694,-179.692,6.096,149.005
C00576=1166.105,40.596,-48.678,-179.694,6.096,149.006
C00577=1166.110,40.347,-48.663,-179.697,6.094,149.006
C00578=1166.115,40.097,-48.648,-179.700,6.093,149.007
C00579=1166.120,39.848,-48.633,-179.702,6.093,149.007
C00580=1166.125,39.599,-48.617,-179.705,6.091,149.008
C00581=1166.131,39.349,-48.602,-179.707,6.090,149.008
C00582=1166.135,39.099,-48.587,-179.710,6.090,149.009
C00583=1166.141,38.850,-48.571,-179.712,6.089,149.009
C00584=1166.145,38.601,-48.556,-179.715,6.088,149.010
C00585=1166.151,38.351,-48.541,-179.717,6.087,149.011
C00586=1166.156,38.101,-48.526,-179.720,6.086,149.011
C00587=1166.161,37.852,-48.511,-179.723,6.085,149.012
C00588=1166.166,37.603,-48.496,-179.725,6.084,149.012
C00589=1166.170,37.353,-48.480,-179.728,6.084,149.013
C00590=1166.175,37.103,-48.466,-179.730,6.083,149.013
C00591=1166.181,36.854,-48.450,-179.733,6.082,149.014
C00592=1166.185,36.605,-48.435,-179.736,6.081,149.015
C00593=1166.191,36.355,-48.419,-179.738,6.080,149.015
C00594=1166.196,36.106,-48.405,-179.740,6.079,149.016
C00595=1166.201,35.856,-48.389,-179.744,6.078,149.016
C00596=1166.206,35.607,-48.374,-179.746,6.077,149.017
C00597=1166.211,35.357,-48.360,-179.748,6.077,149.018
C00598=1166.216,35.108,-48.345,-179.751,6.075,149.018
C00599=1166.221,34.859,-48.329,-179.754,6.075,149.019
C00600=1166.226,34.608,-48.314,-179.756,6.074,149.019
C00601=1166.231,34.359,-48.299,-179.759,6.073,149.020
C00602=1166.236,34.110,-48.284,-179.762,6.072,149.020
C00603=1166.241,33.860,-48.270,-179.764,6.071,149.021
C00604=1166.246,33.611,-48.254,-179.767,6.071,149.022
C00605=1166.251,33.361,-48.240,-179.769,6.070,149.022
C00606=1166.257,33.111,-48.224,-179.772,6.069,149.023
C00607=1166.261,32.862,-48.209,-179.774,6.068,149.023
C00608=1166.266,32.613,-48.195,-179.777,6.067,149.024
C00609=1166.272,32.363,-48.179,-179.779,6.066,149.024
C00610=1166.277,32.113,-48.165,-179.782,6.065,149.025
C00611=1166.281,31.864,-48.150,-179.784,6.064,149.025
C00612=1166.287,31.614,-48.135,-179.787,6.064,149.026
C00613=1166.291,31.365,-48.120,-179.790,6.063,149.027
C00614=1166.297,31.116,-48.105,-179.792,6.062,149.027
C00615=1166.302,30.866,-48.090,-179.795,6.061,149.028
C00616=1166.306,30.617,-48.075,-179.797,6.060,149.028
C00617=1166.312,30.367,-48.060,-179.800,6.060,149.029
C00618=1166.317,30.118,-48.045,-179.803,6.058,149.029
C00619=1166.322,29.868,-48.031,-179.805,6.058,149.030
C00620=1166.327,29.619,-48.016,-179.807,6.057,149.031
C00621=1166.332,29.369,-48.001,-179.810,6.056,149.031
C00622=1166.337,29.119,-47.987,-179.813,6.056,149.032
C00623=1166.342,28.870,-47.972,-179.815,6.054,149.032
C00624=1166.347,28.620,-47.957,-179.818,6.054,149.033
C00625=1166.353,28.352,-47.941,-179.820,6.053,149.034
C00626=1166.358,28.083,-47.926,-179.824,6.052,149.034
C00627=1166.364,27.814,-47.909,-179.826,6.051,149.035
C00628=1166.369,27.545,-47.894,-179.829,6.051,149.036
C00629=1166.373,27.296,-47.879,-179.832,6.049,149.036
C00630=1166.379,27.046,-47.864,-179.834,6.049,149.037
C00631=1166.384,26.796,-47.850,-179.836,6.048,149.037
C00632=1166.389,26.547,-47.835,-179.839,6.047,149.038
C00633=1166.394,26.297,-47.820,-179.842,6.046,149.038
C00634=1166.399,26.047,-47.805,-179.844,6.045,149.039
C00635=1166.404,25.798,-47.790,-179.847,6.045,149.040
C00636=1166.409,25.549,-47.776,-179.849,6.044,149.040
C00637=1166.414,25.299,-47.762,-179.852,6.043,149.041
C00638=1166.419,25.050,-47.747,-179.855,6.042,149.041
C00639=1166.425,24.800,-47.732,-179.857,6.041,149.042
C00640=1166.430,24.551,-47.718,-179.859,6.040,149.042
C00641=1166.434,24.301,-47.703,-179.862,6.040,149.043
C00642=1166.439,24.052,-47.689,-179.864,6.039,149.043
C00643=1166.444,23.802,-47.675,-179.867,6.038,149.044
C00644=1166.449,23.552,-47.660,-179.870,6.037,149.045
C00645=1166.455,23.303,-47.645,-179.872,6.036,149.045
C00646=1166.460,23.053,-47.630,-179.875,6.036,149.046
C00647=1166.465,22.804,-47.616,-179.877,6.035,149.046
C00648=1166.470,22.554,-47.602,-179.880,6.034,149.047
C00649=1166.475,22.305,-47.587,-179.883,6.033,149.048
C00650=1166.480,22.056,-47.573,-179.885,6.032,149.048
C00651=1166.485,21.806,-47.559,-179.888,6.032,149.049
C00652=1166.490,21.556,-47.544,-179.890,6.031,149.049
C00653=1166.495,21.306,-47.529,-179.893,6.031,149.050
C00654=1166.500,21.057,-47.514,-179.895,6.029,149.050
C00655=1166.505,20.808,-47.501,-179.898,6.029,149.051
C00656=1166.510,20.558,-47.486,-179.900,6.028,149.052
C00657=1166.515,20.309,-47.472,-179.903,6.027,149.052
C00658=1166.520,20.059,-47.458,-179.905,6.027,149.053
C00659=1166.525,19.809,-47.443,-179.908,6.026,149.053
C00660=1166.530,19.560,-47.429,-179.911,6.025,149.054
C00661=1166.536,19.311,-47.415,-179.913,6.024,149.055
C00662=1166.540,19.062,-47.400,-179.916,6.023,149.055
C00663=1166.545,18.812,-47.386,-179.918,6.023,149.056
C00664=1166.550,18.562,-47.372,-179.921,6.022,149.056
C00665=1166.556,18.312,-47.357,-179.923,6.022,149.057
C00666=1166.562,18.063,-47.343,-179.926,6.020,149.058
C00667=1166.567,17.813,-47.329,-179.929,6.019,149.058
C00668=1166.572,17.564,-47.314,-179.931,6.019,149.059
C00669=1166.576,17.314,-47.300,-179.933,6.018,149.059
C00670=1166.581,17.064,-47.286,-179.936,6.017,149.060
C00671=1166.587,16.815,-47.272,-179.938,6.017,149.060
C00672=1166.592,16.565,-47.258,-179.941,6.016,149.061
C00673=1166.597,16.316,-47.243,-179.944,6.015,149.062
C00674=1166.602,16.066,-47.229,-179.946,6.014,149.062
C00675=1166.606,15.817,-47.215,-179.948,6.013,149.063
C00676=1166.612,15.568,-47.202,-179.951,6.013,149.063
C00677=1166.617,15.318,-47.187,-179.953,6.012,149.064
C00678=1166.622,15.068,-47.173,-179.956,6.012,149.065
C00679=1166.627,14.819,-47.159,-179.959,6.010,149.065
C00680=1166.632,14.570,-47.145,-179.961,6.010,149.066
C00681=1166.637,14.320,-47.130,-179.964,6.009,149.066
C00682=1166.642,14.070,-47.116,-179.966,6.008,149.067
C00683=1166.647,13.820,-47.102,-179.969,6.008,149.068
C00684=1166.652,13.571,-47.088,-179.971,6.007,149.068
C00685=1166.657,13.322,-47.074,-179.974,6.006,149.069
C00686=1166.663,13.071,-47.060,-179.977,6.005,149.069
C00687=1166.668,12.822,-47.046,-179.979,6.004,149.070
C00688=1166.673,12.573,-47.032,-179.982,6.004,149.071
C00689=1166.677,12.323,-47.018,-179.984,6.003,149.071
C00690=1166.682,12.073,-47.004,-179.986,6.003,149.072
C00691=1166.688,11.824,-46.990,-179.989,6.002,149.072
C00692=1166.693,11.575,-46.976,-179.991,6.001,149.073
C00693=1166.698,11.324,-46.962,-179.994,6.001,149.074
C00694=1166.704,11.075,-46.948,-179.997,5.999,149.074
C00695=1166.709,10.826,-46.934,-179.999,5.999,149.075
C00696=1166.714,10.576,-46.920,179.998,5.998,149.075
C00697=1166.718,10.327,-46.906,179.996,5.997,149.076
C00698=1166.723,10.078,-46.892,179.993,5.997,149.076
C00699=1166.729,9.827,-46.879,179.991,5.996,149.077
C00700=1166.734,9.578,-46.865,179.988,5.996,149.078
C00701=1166.739,9.329,-46.850,179.986,5.995,149.078
C00702=1166.743,9.079,-46.837,179.984,5.994,149.079
C00703=1166.749,8.830,-46.824,179.980,5.993,149.079
C00704=1166.754,8.580,-46.809,179.978,5.992,149.080
C00705=1166.759,8.330,-46.795,179.975,5.992,149.081
C00706=1166.765,8.081,-46.781,179.973,5.991,149.081
C00707=1166.769,7.831,-46.768,179.971,5.990,149.082
C00708=1166.774,7.581,-46.754,179.968,5.990,149.082
C00709=1166.780,7.332,-46.740,179.966,5.989,149.083
C00710=1166.785,7.082,-46.726,179.963,5.989,149.084
C00711=1166.790,6.832,-46.712,179.961,5.988,149.084
C00712=1166.795,6.584,-46.699,179.958,5.987,149.085
C00713=1166.800,6.333,-46.685,179.956,5.986,149.085
C00714=1166.806,6.084,-46.671,179.953,5.985,149.086
C00715=1166.810,5.835,-46.658,179.950,5.985,149.087
C00716=1166.815,5.585,-46.644,179.948,5.984,149.087
C00717=1166.821,5.336,-46.630,179.945,5.984,149.088
C00718=1166.826,5.086,-46.616,179.943,5.983,149.088
C00719=1166.831,4.837,-46.603,179.941,5.982,149.089
C00720=1166.836,4.587,-46.589,179.938,5.982,149.090
C00721=1166.841,4.336,-46.575,179.936,5.981,149.090
C00722=1166.846,4.088,-46.562,179.933,5.981,149.091
C00723=1166.851,3.838,-46.548,179.931,5.980,149.091
C00724=1166.857,3.588,-46.535,179.928,5.978,149.092
C00725=1166.861,3.339,-46.521,179.926,5.978,149.092
C00726=1166.867,3.089,-46.508,179.923,5.977,149.093
C00727=1166.872,2.840,-46.494,179.920,5.977,149.094
C00728=1166.876,2.590,-46.481,179.918,5.976,149.094
C00729=1166.882,2.321,-46.466,179.915,5.975,149.095
C00730=1166.888,2.052,-46.451,179.913,5.975,149.095
C00731=1166.893,1.782,-46.436,179.910,5.974,149.096
C00732=1166.899,1.512,-46.422,179.907,5.973,149.097
C00733=1166.904,1.263,-46.408,179.905,5.972,149.097
C00734=1166.909,1.013,-46.395,179.902,5.972,149.098
C00735=1166.914,0.764,-46.381,179.900,5.971,149.098
C00736=1166.919,0.514,-46.368,179.897,5.971,149.099
C00737=1166.924,0.265,-46.354,179.895,5.970,149.100
C00738=1166.929,0.015,-46.341,179.892,5.969,149.100
C00739=1166.935,-0.234,-46.327,179.890,5.969,149.101
C00740=1166.939,-0.484,-46.314,179.888,5.968,149.101
C00741=1166.945,-0.733,-46.300,179.885,5.968,149.102
C00742=1166.950,-0.983,-46.287,179.883,5.967,149.103
C00743=1166.955,-1.233,-46.274,179.880,5.966,149.103
C00744=1166.960,-1.482,-46.260,179.877,5.966,149.104
C00745=1166.965,-1.732,-46.247,179.875,5.965,149.104
C00746=1166.970,-1.981,-46.233,179.872,5.964,149.105
C00747=1166.975,-2.231,-46.220,179.870,5.963,149.106
C00748=1166.980,-2.481,-46.207,179.867,5.963,149.106
C00749=1166.985,-2.730,-46.193,179.865,5.962,149.107
C00750=1166.990,-2.980,-46.180,179.862,5.961,149.107
C00751=1166.996,-3.229,-46.167,179.860,5.961,149.108
C00752=1167.001,-3.478,-46.153,179.858,5.960,149.109
C00753=1167.006,-3.728,-46.140,179.855,5.960,149.109
C00754=1167.012,-3.978,-46.127,179.852,5.959,149.110
C00755=1167.016,-4.227,-46.114,179.850,5.958,149.110
C00756=1167.022,-4.477,-46.100,179.847,5.958,149.111
C00757=1167.026,-4.727,-46.087,179.845,5.957,149.112
C00758=1167.032,-4.976,-46.073,179.843,5.957,149.112
C00759=1167.036,-5.226,-46.060,179.840,5.956,149.113
C00760=1167.042,-5.476,-46.047,179.838,5.955,149.113
C00761=1167.047,-5.725,-46.035,179.835,5.955,149.114
C00762=1167.052,-5.975,-46.020,179.833,5.954,149.115
C00763=1167.057,-6.224,-46.008,179.830,5.954,149.115
C00764=1167.063,-6.474,-45.994,179.828,5.953,149.116
C00765=1167.068,-6.724,-45.982,179.825,5.952,149.116
C00766=1167.073,-6.973,-45.967,179.823,5.952,149.117
C00767=1167.078,-7.223,-45.955,179.821,5.951,149.118
C00768=1167.083,-7.472,-45.942,179.818,5.951,149.118
C00769=1167.088,-7.722,-45.929,179.816,5.950,149.119
C00770=1167.093,-7.972,-45.916,179.813,5.949,149.119
C00771=1167.098,-8.221,-45.902,179.810,5.949,149.120
C00772=1167.103,-8.471,-45.889,179.808,5.948,149.121
C00773=1167.108,-8.720,-45.877,179.806,5.948,149.121
C00774=1167.114,-8.970,-45.863,179.803,5.947,149.122
C00775=1167.119,-9.220,-45.850,179.801,5.946,149.122
C00776=1167.124,-9.469,-45.838,179.798,5.946,149.123
C00777=1167.129,-9.719,-45.824,179.796,5.945,149.124
C00778=1167.134,-9.968,-45.811,179.793,5.945,149.124
C00779=1167.139,-10.218,-45.797,179.791,5.944,149.125
C00780=1167.144,-10.468,-45.785,179.788,5.943,149.125
C00781=1167.150,-10.717,-45.772,179.786,5.943,149.126
C00782=1167.155,-10.967,-45.759,179.784,5.942,149.127
C00783=1167.160,-11.217,-45.746,179.781,5.942,149.127
C00784=1167.165,-11.466,-45.733,179.779,5.941,149.128
C00785=1167.170,-11.716,-45.720,179.776,5.940,149.128
C00786=1167.175,-11.966,-45.707,179.773,5.940,149.129
C00787=1167.181,-12.215,-45.695,179.771,5.939,149.130
C00788=1167.185,-12.465,-45.682,179.769,5.939,149.130
C00789=1167.191,-12.715,-45.668,179.766,5.938,149.131
C00790=1167.196,-12.964,-45.656,179.764,5.937,149.131
C00791=1167.201,-13.214,-45.643,179.761,5.937,149.132
C00792=1167.206,-13.464,-45.630,179.759,5.936,149.133
C00793=1167.212,-13.713,-45.617,179.756,5.936,149.133
C00794=1167.217,-13.962,-45.604,179.754,5.935,149.134
C00795=1167.221,-14.212,-45.592,179.751,5.934,149.135
C00796=1167.227,-14.462,-45.578,179.749,5.934,149.135
C00797=1167.232,-14.711,-45.566,179.747,5.933,149.136
C00798=1167.237,-14.961,-45.553,179.744,5.933,149.136
C00799=1167.242,-15.211,-45.540,179.742,5.932,149.137
C00800=1167.248,-15.460,-45.527,179.739,5.931,149.138
C00801=1167.253,-15.709,-45.514,179.736,5.931,149.138
C00802=1167.257,-15.959,-45.501,179.734,5.930,149.139
C00803=1167.263,-16.209,-45.489,179.732,5.930,149.139
C00804=1167.268,-16.458,-45.476,179.729,5.929,149.140
C00805=1167.273,-16.708,-45.463,179.727,5.928,149.141
C00806=1167.278,-16.958,-45.450,179.724,5.928,149.141
C00807=1167.283,-17.207,-45.437,179.722,5.927,149.142
C00808=1167.289,-17.457,-45.426,179.719,5.927,149.142
C00809=1167.294,-17.706,-45.413,179.717,5.926,149.143
C00810=1167.299,-17.957,-45.399,179.714,5.925,149.144
C00811=1167.304,-18.206,-45.387,179.712,5.925,149.144
C00812=1167.309,-18.455,-45.374,179.710,5.924,149.145
C00813=1167.314,-18.705,-45.362,179.708,5.925,149.145
C00814=1167.319,-18.955,-45.349,179.705,5.924,149.146
C00815=1167.324,-19.205,-45.337,179.703,5.923,149.147
C00816=1167.330,-19.454,-45.324,179.700,5.923,149.147
C00817=1167.335,-19.704,-45.311,179.698,5.922,149.148
C00818=1167.340,-19.953,-45.298,179.695,5.922,149.148
C00819=1167.345,-20.203,-45.285,179.693,5.921,149.149
C00820=1167.350,-20.453,-45.273,179.690,5.920,149.150
C00821=1167.355,-20.702,-45.261,179.688,5.920,149.150
C00822=1167.361,-20.951,-45.248,179.686,5.919,149.151
C00823=1167.366,-21.201,-45.236,179.683,5.919,149.151
C00824=1167.371,-21.452,-45.223,179.681,5.918,149.152
C00825=1167.376,-21.701,-45.210,179.678,5.917,149.153
C00826=1167.382,-21.950,-45.198,179.676,5.917,149.153
C00827=1167.387,-22.200,-45.185,179.673,5.916,149.154
C00828=1167.392,-22.450,-45.173,179.671,5.916,149.154
C00829=1167.397,-22.699,-45.161,179.668,5.915,149.155
C00830=1167.402,-22.949,-45.148,179.666,5.915,149.156
C00831=1167.407,-23.199,-45.136,179.664,5.914,149.156
C00832=1167.412,-23.448,-45.123,179.661,5.914,149.157
C00833=1167.417,-23.718,-45.109,179.659,5.914,149.158
C00834=1167.424,-23.988,-45.096,179.656,5.912,149.158
C00835=1167.429,-24.258,-45.083,179.653,5.911,149.159
C00836=1167.435,-24.527,-45.070,179.651,5.911,149.159
C00837=1167.439,-24.777,-45.057,179.648,5.911,149.160
C00838=1167.444,-25.027,-45.044,179.646,5.910,149.161
C00839=1167.450,-25.277,-45.032,179.644,5.910,149.161
C00840=1167.455,-25.526,-45.020,179.641,5.910,149.162
C00841=1167.460,-25.775,-45.007,179.639,5.909,149.162
C00842=1167.466,-26.025,-44.995,179.636,5.908,149.163
C00843=1167.471,-26.274,-44.983,179.634,5.908,149.164
C00844=1167.476,-26.524,-44.971,179.631,5.907,149.164
C00845=1167.481,-26.774,-44.958,179.629,5.907,149.165
C00846=1167.486,-27.024,-44.945,179.627,5.906,149.165
C00847=1167.491,-27.274,-44.933,179.624,5.906,149.166
C00848=1167.496,-27.523,-44.921,179.622,5.905,149.167
C00849=1167.502,-27.773,-44.909,179.619,5.904,149.167
C00850=1167.507,-28.022,-44.896,179.617,5.905,149.168
C00851=1167.512,-28.272,-44.884,179.615,5.904,149.168
C00852=1167.517,-28.521,-44.872,179.612,5.903,149.169
C00853=1167.523,-28.771,-44.860,179.610,5.903,149.170
C00854=1167.528,-29.021,-44.847,179.607,5.902,149.170
C00855=1167.533,-29.271,-44.836,179.605,5.902,149.171
C00856=1167.538,-29.521,-44.823,179.603,5.901,149.172
C00857=1167.543,-29.771,-44.811,179.600,5.900,149.172
C00858=1167.548,-30.020,-44.799,179.598,5.900,149.173
C00859=1167.553,-30.270,-44.787,179.595,5.899,149.173
C00860=1167.558,-30.519,-44.774,179.593,5.900,149.174
C00861=1167.564,-30.769,-44.762,179.591,5.899,149.175
C00862=1167.569,-31.018,-44.750,179.588,5.898,149.175
C00863=1167.574,-31.268,-44.738,179.586,5.898,149.176
C00864=1167.579,-31.517,-44.725,179.583,5.897,149.176
C00865=1167.585,-31.767,-44.713,179.581,5.896,149.177
C00866=1167.590,-32.017,-44.701,179.578,5.896,149.178
C00867=1167.595,-32.266,-44.689,179.576,5.895,149.178
C00868=1167.600,-32.516,-44.678,179.574,5.895,149.179
C00869=1167.605,-32.765,-44.665,179.572,5.895,149.179
C00870=1167.611,-33.015,-44.653,179.569,5.894,149.180
C00871=1167.616,-33.265,-44.641,179.567,5.894,149.181
C00872=1167.621,-33.515,-44.629,179.564,5.893,149.181
C00873=1167.626,-33.764,-44.617,179.562,5.893,149.182
C00874=1167.631,-34.014,-44.605,179.559,5.892,149.182
C00875=1167.636,-34.264,-44.593,179.557,5.891,149.183
C00876=1167.642,-34.514,-44.581,179.554,5.891,149.184
C00877=1167.647,-34.763,-44.569,179.552,5.891,149.184
C00878=1167.652,-35.012,-44.557,179.550,5.890,149.185
C00879=1167.657,-35.262,-44.545,179.547,5.890,149.186
C00880=1167.663,-35.512,-44.533,179.545,5.889,149.186
C00881=1167.668,-35.762,-44.521,179.543,5.889,149.187
C00882=1167.673,-36.012,-44.509,179.540,5.888,149.187
C00883=1167.678,-36.261,-44.497,179.538,5.888,149.188
C00884=1167.683,-36.511,-44.485,179.535,5.887,149.189
C00885=1167.688,-36.760,-44.473,179.533,5.887,149.189
C00886=1167.694,-37.010,-44.461,179.531,5.887,149.190
C00887=1167.698,-37.260,-44.450,179.529,5.886,149.190
C00888=1167.704,-37.509,-44.437,179.526,5.885,149.191
C00889=1167.710,-37.759,-44.426,179.523,5.885,149.192
C00890=1167.715,-38.009,-44.414,179.521,5.884,149.192
C00891=1167.720,-38.258,-44.403,179.518,5.884,149.193
C00892=1167.725,-38.508,-44.391,179.517,5.884,149.193
C00893=1167.730,-38.757,-44.378,179.514,5.883,149.194
C00894=1167.735,-39.007,-44.367,179.512,5.883,149.195
C00895=1167.740,-39.257,-44.355,179.509,5.882,149.195
C00896=1167.746,-39.507,-44.343,179.507,5.882,149.196
C00897=1167.751,-39.757,-44.331,179.504,5.881,149.196
C00898=1167.756,-40.006,-44.319,179.502,5.881,149.197
C00899=1167.761,-40.256,-44.307,179.500,5.880,149.197
C00900=1167.767,-40.505,-44.296,179.498,5.880,149.198
C00901=1167.772,-40.755,-44.284,179.495,5.880,149.199
C00902=1167.777,-41.005,-44.272,179.493,5.879,149.199
C00903=1167.783,-41.254,-44.261,179.490,5.878,149.200
C00904=1167.787,-41.504,-44.249,179.488,5.878,149.201
C00905=1167.793,-41.753,-44.237,179.486,5.878,149.201
C00906=1167.797,-42.003,-44.225,179.484,5.877,149.202
C00907=1167.803,-42.253,-44.214,179.481,5.877,149.202
C00908=1167.808,-42.503,-44.202,179.478,5.876,149.203
C00909=1167.813,-42.752,-44.191,179.476,5.875,149.204
C00910=1167.819,-43.002,-44.179,179.474,5.876,149.204
C00911=1167.824,-43.252,-44.167,179.472,5.875,149.205
C00912=1167.829,-43.501,-44.156,179.469,5.875,149.205
C00913=1167.834,-43.751,-44.144,179.467,5.874,149.206
C00914=1167.839,-44.001,-44.132,179.464,5.873,149.207
C00915=1167.844,-44.251,-44.121,179.462,5.873,149.207
C00916=1167.850,-44.500,-44.109,179.460,5.873,149.208
C00917=1167.855,-44.750,-44.098,179.457,5.873,149.209
C00918=1167.861,-45.000,-44.086,179.455,5.872,149.209
C00919=1167.865,-45.249,-44.075,179.453,5.871,149.210
C00920=1167.871,-45.499,-44.063,179.450,5.871,149.210
C00921=1167.875,-45.749,-44.051,179.448,5.870,149.211
C00922=1167.881,-45.998,-44.040,179.446,5.870,149.212
C00923=1167.887,-46.248,-44.028,179.443,5.870,149.212
C00924=1167.892,-46.498,-44.017,179.441,5.869,149.213
C00925=1167.897,-46.748,-44.005,179.439,5.868,149.213
C00926=1167.902,-46.997,-43.994,179.436,5.868,149.214
C00927=1167.908,-47.246,-43.982,179.434,5.868,149.215
C00928=1167.912,-47.496,-43.971,179.432,5.868,149.215
C00929=1167.918,-47.746,-43.959,179.429,5.867,149.216
C00930=1167.923,-47.996,-43.948,179.427,5.866,149.216
C00931=1167.928,-48.246,-43.936,179.424,5.866,149.217
C00932=1167.933,-48.494,-43.925,179.423,5.866,149.217
C00933=1167.939,-48.744,-43.913,179.420,5.866,149.218
C00934=1167.943,-48.994,-43.902,179.417,5.865,149.219
C00935=1167.949,-49.244,-43.890,179.415,5.864,149.219
C00936=1167.954,-49.494,-43.880,179.412,5.864,149.220
C00937=1167.960,-49.764,-43.867,179.410,5.863,149.221
C00938=1167.965,-50.035,-43.854,179.408,5.863,149.221
C00939=1167.971,-50.305,-43.842,179.405,5.863,149.222
C00940=1167.977,-50.575,-43.829,179.403,5.863,149.223
C00941=1167.982,-50.825,-43.818,179.401,5.862,149.223
C00942=1167.988,-51.074,-43.807,179.398,5.861,149.224
C00943=1167.993,-51.325,-43.796,179.395,5.861,149.225
C00944=1167.998,-51.575,-43.784,179.393,5.860,149.225
C00945=1168.003,-51.824,-43.773,179.391,5.861,149.226
C00946=1168.008,-52.073,-43.762,179.389,5.860,149.226
C00947=1168.013,-52.323,-43.750,179.386,5.859,149.227
C00948=1168.018,-52.573,-43.740,179.384,5.859,149.227
C00949=1168.024,-52.823,-43.728,179.381,5.858,149.228
C00950=1168.029,-53.072,-43.717,179.380,5.858,149.229
C00951=1168.034,-53.322,-43.705,179.377,5.858,149.229
C00952=1168.039,-53.572,-43.694,179.374,5.857,149.230
C00953=1168.045,-53.821,-43.683,179.372,5.857,149.230
C00954=1168.050,-54.071,-43.671,179.370,5.857,149.231
C00955=1168.055,-54.321,-43.660,179.368,5.856,149.232
C00956=1168.060,-54.570,-43.649,179.365,5.856,149.232
C00957=1168.066,-54.820,-43.638,179.363,5.855,149.233
C00958=1168.071,-55.070,-43.627,179.361,5.855,149.233
C00959=1168.075,-55.320,-43.615,179.359,5.855,149.234
C00960=1168.082,-55.569,-43.605,179.356,5.854,149.235
C00961=1168.086,-55.819,-43.593,179.354,5.854,149.235
C00962=1168.091,-56.069,-43.582,179.351,5.853,149.236
C00963=1168.097,-56.318,-43.571,179.349,5.853,149.237
C00964=1168.102,-56.568,-43.560,179.347,5.852,149.237
C00965=1168.107,-56.818,-43.549,179.344,5.852,149.238
C00966=1168.113,-57.068,-43.538,179.342,5.851,149.238
C00967=1168.118,-57.317,-43.527,179.340,5.852,149.239
C00968=1168.123,-57.567,-43.515,179.338,5.851,149.239
C00969=1168.128,-57.816,-43.505,179.335,5.850,149.240
C00970=1168.134,-58.066,-43.493,179.333,5.850,149.241
C00971=1168.138,-58.316,-43.482,179.331,5.850,149.241
C00972=1168.144,-58.565,-43.472,179.328,5.850,149.242
C00973=1168.149,-58.815,-43.460,179.326,5.849,149.242
C00974=1168.154,-59.065,-43.449,179.323,5.848,149.243
C00975=1168.160,-59.315,-43.438,179.322,5.848,149.244
C00976=1168.164,-59.564,-43.427,179.319,5.848,149.244
C00977=1168.170,-59.815,-43.416,179.317,5.847,149.245
C00978=1168.175,-60.064,-43.405,179.314,5.847,149.246
C00979=1168.180,-60.314,-43.394,179.312,5.847,149.246
C00980=1168.186,-60.563,-43.383,179.310,5.846,149.247
C00981=1168.191,-60.813,-43.372,179.307,5.846,149.247
C00982=1168.196,-61.063,-43.361,179.305,5.845,149.248
C00983=1168.201,-61.312,-43.350,179.303,5.846,149.249
C00984=1168.206,-61.562,-43.339,179.301,5.845,149.249
C00985=1168.212,-61.811,-43.329,179.298,5.844,149.250
C00986=1168.217,-62.062,-43.317,179.296,5.844,149.250
C00987=1168.222,-62.311,-43.306,179.294,5.844,149.251
C00988=1168.228,-62.561,-43.296,179.292,5.843,149.251
C00989=1168.232,-62.810,-43.285,179.289,5.843,149.252
C00990=1168.238,-63.060,-43.274,179.287,5.842,149.253
C00991=1168.243,-63.310,-43.263,179.285,5.842,149.253
C00992=1168.249,-63.560,-43.252,179.282,5.842,149.254
C00993=1168.254,-63.809,-43.241,179.280,5.841,149.255
C00994=1168.259,-64.059,-43.230,179.277,5.841,149.255
C00995=1168.264,-64.309,-43.220,179.276,5.841,149.256
C00996=1168.269,-64.559,-43.209,179.273,5.840,149.256
C00997=1168.275,-64.808,-43.198,179.271,5.840,149.257
C00998=1168.280,-65.058,-43.187,179.269,5.840,149.258
C00999=1168.286,-65.308,-43.177,179.267,5.839,149.258
C01000=1168.290,-65.557,-43.165,179.264,5.839,149.259
C01001=1168.296,-65.807,-43.155,179.262,5.838,149.259
C01002=1168.301,-66.057,-43.145,179.260,5.838,149.260
C01003=1168.306,-66.307,-43.133,179.258,5.838,149.260
C01004=1168.312,-66.556,-43.122,179.255,5.837,149.261
C01005=1168.317,-66.806,-43.111,179.253,5.838,149.262
C01006=1168.322,-67.056,-43.101,179.251,5.837,149.262
C01007=1168.327,-67.306,-43.090,179.248,5.836,149.263
C01008=1168.332,-67.555,-43.079,179.246,5.836,149.264
C01009=1168.337,-67.805,-43.069,179.244,5.836,149.264
C01010=1168.343,-68.055,-43.059,179.242,5.835,149.265
C01011=1168.348,-68.304,-43.047,179.239,5.835,149.265
C01012=1168.353,-68.554,-43.037,179.237,5.835,149.266
C01013=1168.358,-68.804,-43.027,179.235,5.834,149.267
C01014=1168.364,-69.053,-43.016,179.232,5.834,149.267
C01015=1168.369,-69.304,-43.005,179.230,5.833,149.268
C01016=1168.375,-69.553,-42.994,179.228,5.833,149.268
C01017=1168.380,-69.803,-42.984,179.225,5.833,149.269
C01018=1168.385,-70.052,-42.973,179.223,5.832,149.269
C01019=1168.391,-70.302,-42.963,179.221,5.832,149.270
C01020=1168.396,-70.552,-42.952,179.219,5.832,149.271
C01021=1168.401,-70.801,-42.941,179.216,5.831,149.271
C01022=1168.406,-71.051,-42.931,179.214,5.831,149.272
C01023=1168.412,-71.301,-42.920,179.212,5.831,149.273
C01024=1168.417,-71.551,-42.910,179.209,5.830,149.273
C01025=1168.422,-71.801,-42.900,179.207,5.830,149.274
C01026=1168.427,-72.050,-42.888,179.205,5.830,149.274
C01027=1168.433,-72.300,-42.878,179.203,5.829,149.275
C01028=1168.438,-72.550,-42.867,179.200,5.829,149.276
C01029=1168.443,-72.799,-42.857,179.199,5.829,149.276
C01030=1168.449,-73.048,-42.846,179.196,5.828,149.277
C01031=1168.454,-73.299,-42.836,179.194,5.828,149.277
C01032=1168.459,-73.548,-42.826,179.192,5.828,149.278
C01033=1168.464,-73.798,-42.815,179.190,5.827,149.279
C01034=1168.470,-74.048,-42.805,179.187,5.827,149.279
C01035=1168.475,-74.298,-42.794,179.185,5.826,149.280
C01036=1168.480,-74.547,-42.783,179.183,5.826,149.280
C01037=1168.486,-74.797,-42.773,179.180,5.826,149.281
C01038=1168.491,-75.047,-42.762,179.178,5.825,149.282
C01039=1168.496,-75.296,-42.752,179.176,5.825,149.282
C01040=1168.501,-75.547,-42.742,179.174,5.825,149.283
C01041=1168.507,-75.817,-42.731,179.171,5.824,149.283
C01042=1168.513,-76.089,-42.720,179.169,5.824,149.284
C01043=1168.518,-76.360,-42.708,179.167,5.824,149.285
C01044=1168.524,-76.630,-42.697,179.164,5.824,149.285
C01045=1168.529,-76.881,-42.686,179.162,5.823,149.286
C01046=1168.535,-77.130,-42.676,179.159,5.823,149.287
C01047=1168.541,-77.380,-42.666,179.157,5.823,149.287
C01048=1168.545,-77.630,-42.656,179.155,5.822,149.288
C01049=1168.550,-77.879,-42.646,179.153,5.821,149.288
C01050=1168.556,-78.129,-42.635,179.151,5.822,149.289
C01051=1168.561,-78.379,-42.625,179.148,5.821,149.289
C01052=1168.567,-78.629,-42.615,179.146,5.821,149.290
C01053=1168.572,-78.878,-42.604,179.144,5.821,149.291
C01054=1168.577,-79.128,-42.594,179.141,5.820,149.291
C01055=1168.583,-79.378,-42.584,179.139,5.819,149.292
C01056=1168.587,-79.628,-42.574,179.137,5.820,149.293
C01057=1168.593,-79.877,-42.563,179.135,5.819,149.293
C01058=1168.598,-80.127,-42.553,179.132,5.819,149.294
C01059=1168.603,-80.377,-42.543,179.131,5.819,149.294
C01060=1168.609,-80.627,-42.532,179.128,5.818,149.295
C01061=1168.614,-80.876,-42.522,179.126,5.817,149.295
C01062=1168.619,-81.126,-42.512,179.124,5.818,149.296
C01063=1168.624,-81.376,-42.502,179.122,5.817,149.297
C01064=1168.630,-81.625,-42.492,179.119,5.818,149.297
C01065=1168.635,-81.876,-42.481,179.117,5.817,149.298
C01066=1168.640,-82.125,-42.471,179.115,5.816,149.298
C01067=1168.646,-82.375,-42.461,179.113,5.816,149.299
C01068=1168.651,-82.624,-42.451,179.111,5.816,149.299
C01069=1168.656,-82.874,-42.441,179.108,5.815,149.300
C01070=1168.662,-83.124,-42.430,179.107,5.815,149.301
C01071=1168.667,-83.373,-42.420,179.104,5.815,149.301
C01072=1168.671,-83.623,-42.410,179.102,5.814,149.302
C01073=1168.677,-83.873,-42.401,179.100,5.814,149.303
C01074=1168.683,-84.123,-42.391,179.097,5.814,149.303
C01075=1168.688,-84.372,-42.380,179.095,5.813,149.304
C01076=1168.693,-84.622,-42.370,179.093,5.813,149.304
C01077=1168.698,-84.872,-42.360,179.090,5.813,149.305
C01078=1168.704,-85.121,-42.350,179.088,5.812,149.305
C01079=1168.709,-85.372,-42.339,179.086,5.812,149.306
C01080=1168.714,-85.621,-42.330,179.084,5.812,149.307
C01081=1168.720,-85.871,-42.320,179.082,5.812,149.307
C01082=1168.725,-86.121,-42.310,179.080,5.811,149.308
C01083=1168.730,-86.371,-42.299,179.077,5.811,149.309
C01084=1168.735,-86.620,-42.290,179.075,5.811,149.309
C01085=1168.741,-86.870,-42.280,179.073,5.811,149.310
C01086=1168.747,-87.120,-42.270,179.071,5.810,149.310
C01087=1168.751,-87.370,-42.260,179.069,5.810,149.311
C01088=1168.757,-87.619,-42.250,179.066,5.809,149.311
C01089=1168.762,-87.869,-42.240,179.064,5.809,149.312
C01090=1168.767,-88.118,-42.230,179.062,5.809,149.313
C01091=1168.772,-88.369,-42.220,179.060,5.808,149.313
C01092=1168.778,-88.618,-42.210,179.058,5.809,149.314
C01093=1168.783,-88.868,-42.200,179.056,5.808,149.314
C01094=1168.788,-89.117,-42.190,179.053,5.807,149.315
C01095=1168.794,-89.368,-42.180,179.051,5.807,149.315
C01096=1168.798,-89.617,-42.171,179.049,5.807,149.316
C01097=1168.804,-89.867,-42.161,179.046,5.806,149.317
C01098=1168.810,-90.116,-42.150,179.044,5.807,149.317
C01099=1168.815,-90.366,-42.141,179.042,5.806,149.318
C01100=1168.820,-90.616,-42.131,179.040,5.806,149.319
C01101=1168.825,-90.866,-42.121,179.038,5.806,149.319
C01102=1168.831,-91.116,-42.112,179.036,5.805,149.320
C01103=1168.836,-91.365,-42.102,179.034,5.805,149.320
C01104=1168.841,-91.615,-42.092,179.031,5.804,149.321
C01105=1168.846,-91.866,-42.082,179.029,5.805,149.321
C01106=1168.852,-92.115,-42.072,179.027,5.804,149.322
C01107=1168.857,-92.364,-42.062,179.025,5.804,149.323
C01108=1168.863,-92.614,-42.053,179.023,5.804,149.323
C01109=1168.868,-92.864,-42.043,179.020,5.803,149.324
C01110=1168.873,-93.113,-42.033,179.019,5.803,149.324
C01111=1168.878,-93.364,-42.024,179.016,5.803,149.325
C01112=1168.883,-93.613,-42.014,179.014,5.802,149.325
C01113=1168.889,-93.863,-42.003,179.012,5.802,149.326
C01114=1168.894,-94.113,-41.994,179.010,5.802,149.327
C01115=1168.900,-94.362,-41.984,179.007,5.801,149.327
C01116=1168.905,-94.612,-41.975,179.005,5.801,149.328
C01117=1168.910,-94.862,-41.965,179.003,5.801,149.328
C01118=1168.915,-95.112,-41.955,179.001,5.801,149.329
C01119=1168.921,-95.362,-41.946,178.999,5.800,149.330
C01120=1168.926,-95.611,-41.935,178.996,5.800,149.330
C01121=1168.931,-95.861,-41.927,178.995,5.800,149.331
C01122=1168.937,-96.111,-41.916,178.992,5.799,149.331
C01123=1168.942,-96.361,-41.907,178.990,5.800,149.332
C01124=1168.948,-96.610,-41.897,178.988,5.799,149.332
C01125=1168.953,-96.859,-41.888,178.986,5.799,149.333
C01126=1168.958,-97.110,-41.878,178.984,5.798,149.334
C01127=1168.963,-97.359,-41.868,178.981,5.798,149.334
C01128=1168.969,-97.610,-41.859,178.980,5.798,149.335
C01129=1168.974,-97.859,-41.849,178.977,5.797,149.335
C01130=1168.979,-98.109,-41.840,178.975,5.798,149.336
C01131=1168.984,-98.358,-41.830,178.973,5.797,149.336
C01132=1168.990,-98.608,-41.820,178.970,5.797,149.337
C01133=1168.995,-98.858,-41.811,178.969,5.797,149.338
C01134=1169.001,-99.108,-41.801,178.966,5.796,149.338
C01135=1169.006,-99.357,-41.792,178.965,5.796,149.339
C01136=1169.012,-99.607,-41.782,178.962,5.795,149.339
C01137=1169.017,-99.857,-41.773,178.960,5.795,149.340
C01138=1169.021,-100.107,-41.763,178.958,5.795,149.341
C01139=1169.027,-100.357,-41.754,178.955,5.795,149.341
C01140=1169.032,-100.606,-41.744,178.954,5.795,149.342
C01141=1169.038,-100.857,-41.735,178.951,5.794,149.342
C01142=1169.043,-101.106,-41.725,178.949,5.794,149.343
C01143=1169.049,-101.356,-41.716,178.947,5.794,149.343
C01144=1169.054,-101.606,-41.707,178.945,5.793,149.344
C01145=1169.059,-101.878,-41.696,178.943,5.793,149.345
C01146=1169.065,-102.150,-41.686,178.940,5.793,149.345
C01147=1169.072,-102.421,-41.676,178.938,5.792,149.346
C01148=1169.077,-102.693,-41.666,178.936,5.792,149.347
C01149=1169.082,-102.942,-41.656,178.933,5.792,149.347
C01150=1169.088,-103.192,-41.646,178.931,5.791,149.348
C01151=1169.093,-103.442,-41.637,178.930,5.791,149.348
C01152=1169.098,-103.692,-41.628,178.927,5.791,149.349
C01153=1169.104,-103.942,-41.618,178.925,5.791,149.349
C01154=1169.109,-104.191,-41.609,178.923,5.791,149.350
C01155=1169.114,-104.441,-41.600,178.921,5.791,149.351
C01156=1169.120,-104.691,-41.590,178.919,5.790,149.351
C01157=1169.125,-104.940,-41.581,178.916,5.789,149.352
C01158=1169.130,-105.190,-41.572,178.915,5.789,149.352
C01159=1169.136,-105.440,-41.562,178.912,5.789,149.353
C01160=1169.141,-105.689,-41.553,178.910,5.789,149.354
C01161=1169.146,-105.939,-41.544,178.908,5.788,149.354
C01162=1169.152,-106.189,-41.534,178.906,5.789,149.355
C01163=1169.157,-106.439,-41.526,178.904,5.788,149.355
C01164=1169.162,-106.689,-41.516,178.902,5.788,149.356
C01165=1169.168,-106.939,-41.506,178.900,5.788,149.356
C01166=1169.173,-107.189,-41.498,178.897,5.787,149.357
C01167=1169.178,-107.438,-41.488,178.895,5.787,149.358
C01168=1169.183,-107.688,-41.478,178.893,5.787,149.358
C01169=1169.189,-107.938,-41.470,178.891,5.787,149.359
C01170=1169.194,-108.188,-41.461,178.889,5.786,149.359
C01171=1169.199,-108.437,-41.450,178.887,5.786,149.360
C01172=1169.205,-108.687,-41.442,178.885,5.786,149.360
C01173=1169.210,-108.937,-41.433,178.883,5.786,149.361
C01174=1169.215,-109.187,-41.424,178.880,5.785,149.362
C01175=1169.221,-109.437,-41.414,178.879,5.785,149.362
C01176=1169.226,-109.686,-41.405,178.876,5.785,149.363
C01177=1169.231,-109.936,-41.396,178.874,5.784,149.363
C01178=1169.236,-110.186,-41.387,178.872,5.784,149.364
C01179=1169.242,-110.436,-41.377,178.870,5.784,149.364
C01180=1169.247,-110.686,-41.368,178.868,5.784,149.365
C01181=1169.252,-110.936,-41.360,178.866,5.783,149.366
C01182=1169.257,-111.185,-41.350,178.864,5.784,149.366
C01183=1169.263,-111.435,-41.340,178.861,5.783,149.367
C01184=1169.269,-111.684,-41.332,178.860,5.783,149.367
C01185=1169.274,-111.934,-41.323,178.857,5.783,149.368
C01186=1169.279,-112.184,-41.314,178.856,5.783,149.368
C01187=1169.285,-112.434,-41.305,178.853,5.782,149.369
C01188=1169.290,-112.684,-41.296,178.851,5.782,149.370
C01189=1169.295,-112.933,-41.286,178.849,5.781,149.370
C01190=1169.300,-113.183,-41.277,178.847,5.781,149.371
C01191=1169.305,-113.433,-41.268,178.845,5.781,149.371
C01192=1169.311,-113.683,-41.259,178.843,5.780,149.372
C01193=1169.316,-113.933,-41.250,178.841,5.781,149.373
C01194=1169.322,-114.183,-41.241,178.838,5.780,149.373
C01195=1169.327,-114.432,-41.232,178.837,5.780,149.373
C01196=1169.333,-114.682,-41.224,178.834,5.780,149.374
C01197=1169.338,-114.932,-41.215,178.833,5.780,149.375
C01198=1169.344,-115.182,-41.205,178.830,5.779,149.375
C01199=1169.349,-115.432,-41.196,178.828,5.779,149.376
C01200=1169.354,-115.681,-41.187,178.826,5.779,149.376
C01201=1169.359,-115.931,-41.179,178.824,5.779,149.377
C01202=1169.365,-116.180,-41.170,178.822,5.778,149.378
C01203=1169.370,-116.430,-41.160,178.820,5.778,149.378
C01204=1169.376,-116.680,-41.151,178.818,5.777,149.379
C01205=1169.381,-116.930,-41.142,178.816,5.778,149.379
C01206=1169.386,-117.180,-41.133,178.814,5.777,149.380
C01207=1169.391,-117.429,-41.124,178.812,5.777,149.380
C01208=1169.396,-117.679,-41.115,178.809,5.777,149.381
C01209=1169.402,-117.928,-41.107,178.808,5.777,149.381
C01210=1169.407,-118.178,-41.098,178.806,5.776,149.382
C01211=1169.413,-118.429,-41.090,178.803,5.776,149.383
C01212=1169.418,-118.679,-41.081,178.801,5.776,149.383
C01213=1169.424,-118.929,-41.071,178.799,5.775,149.384
C01214=1169.429,-119.179,-41.062,178.797,5.775,149.384
C01215=1169.435,-119.428,-41.054,178.795,5.775,149.385
C01216=1169.440,-119.678,-41.045,178.793,5.775,149.385
C01217=1169.445,-119.927,-41.036,178.791,5.774,149.386
C01218=1169.450,-120.177,-41.027,178.789,5.774,149.387
C01219=1169.455,-120.427,-41.018,178.787,5.774,149.387
C01220=1169.461,-120.677,-41.009,178.785,5.774,149.388
C01221=1169.466,-120.926,-41.001,178.783,5.773,149.388
C01222=1169.471,-121.176,-40.992,178.781,5.773,149.389
C01223=1169.477,-121.426,-40.983,178.778,5.773,149.389
C01224=1169.482,-121.676,-40.974,178.777,5.773,149.390
C01225=1169.487,-121.926,-40.965,178.774,5.772,149.390
C01226=1169.493,-122.175,-40.957,178.772,5.773,149.391
C01227=1169.498,-122.425,-40.949,178.770,5.772,149.392
C01228=1169.503,-122.675,-40.940,178.769,5.772,149.392
C01229=1169.509,-122.925,-40.931,178.766,5.771,149.393
C01230=1169.514,-123.175,-40.922,178.764,5.771,149.393
C01231=1169.519,-123.424,-40.913,178.762,5.771,149.394
C01232=1169.525,-123.674,-40.904,178.760,5.771,149.394
C01233=1169.530,-123.924,-40.896,178.758,5.770,149.395
C01234=1169.535,-124.174,-40.887,178.756,5.770,149.395
C01235=1169.541,-124.423,-40.879,178.754,5.770,149.396
C01236=1169.546,-124.673,-40.870,178.752,5.770,149.397
C01237=1169.551,-124.923,-40.861,178.750,5.769,149.397
C01238=1169.557,-125.173,-40.853,178.748,5.769,149.398
C01239=1169.563,-125.423,-40.844,178.745,5.769,149.398
C01240=1169.568,-125.672,-40.835,178.744,5.769,149.399
C01241=1169.573,-125.922,-40.826,178.742,5.768,149.399
C01242=1169.578,-126.172,-40.818,178.740,5.769,149.400
C01243=1169.584,-126.422,-40.810,178.737,5.768,149.401
C01244=1169.589,-126.672,-40.801,178.736,5.768,149.401
C01245=1169.595,-126.922,-40.792,178.734,5.767,149.402
C01246=1169.600,-127.171,-40.783,178.732,5.768,149.402
C01247=1169.606,-127.421,-40.775,178.730,5.768,149.403
C01248=1169.611,-127.671,-40.766,178.728,5.767,149.403
C01249=1169.190,-127.682,-40.807,178.724,5.770,149.405
C01250=1169.185,-127.432,-40.816,178.726,5.771,149.405
C01251=1169.179,-127.183,-40.824,178.728,5.771,149.404
C01252=1169.174,-126.933,-40.833,178.730,5.771,149.403
C01253=1169.169,-126.683,-40.842,178.732,5.771,149.403
C01254=1169.162,-126.433,-40.850,178.734,5.772,149.402
C01255=1169.157,-126.183,-40.859,178.736,5.772,149.402
C01256=1169.152,-125.933,-40.868,178.738,5.772,149.401
C01257=1169.147,-125.684,-40.877,178.740,5.772,149.401
C01258=1169.141,-125.434,-40.884,178.742,5.773,149.400
C01259=1169.136,-125.184,-40.893,178.744,5.773,149.399
C01260=1169.131,-124.934,-40.902,178.746,5.773,149.399
C01261=1169.125,-124.684,-40.911,178.748,5.773,149.398
C01262=1169.120,-124.435,-40.920,178.751,5.774,149.398
C01263=1169.114,-124.185,-40.928,178.752,5.774,149.397
C01264=1169.109,-123.935,-40.937,178.755,5.774,149.397
C01265=1169.104,-123.685,-40.946,178.756,5.774,149.396
C01266=1169.099,-123.435,-40.954,178.759,5.775,149.396
C01267=1169.093,-123.186,-40.963,178.760,5.775,149.395
C01268=1169.088,-122.936,-40.972,178.763,5.775,149.395
C01269=1169.083,-122.686,-40.981,178.765,5.775,149.394
C01270=1169.077,-122.436,-40.989,178.767,5.776,149.393
C01271=1169.071,-122.187,-40.997,178.768,5.776,149.393
C01272=1169.066,-121.937,-41.006,178.771,5.776,149.392
C01273=1169.061,-121.687,-41.015,178.773,5.776,149.392
C01274=1169.056,-121.437,-41.024,178.775,5.777,149.391
C01275=1169.051,-121.187,-41.033,178.777,5.776,149.391
C01276=1169.045,-120.938,-41.042,178.779,5.777,149.390
C01277=1169.040,-120.688,-41.050,178.781,5.777,149.390
C01278=1169.035,-120.438,-41.059,178.784,5.778,149.389
C01279=1169.029,-120.188,-41.068,178.785,5.778,149.388
C01280=1169.024,-119.938,-41.076,178.787,5.778,149.388
C01281=1169.018,-119.689,-41.085,178.789,5.778,149.387
C01282=1169.013,-119.439,-41.094,178.792,5.779,149.387
C01283=1169.007,-119.189,-41.103,178.793,5.779,149.386
C01284=1169.002,-118.939,-41.112,178.795,5.779,149.386
C01285=1168.997,-118.689,-41.121,178.797,5.779,149.385
C01286=1168.992,-118.439,-41.130,178.800,5.780,149.384
C01287=1168.986,-118.190,-41.139,178.801,5.780,149.384
C01288=1168.981,-117.940,-41.148,178.804,5.780,149.383
C01289=1168.975,-117.690,-41.156,178.806,5.780,149.383
C01290=1168.970,-117.441,-41.165,178.808,5.781,149.382
C01291=1168.965,-117.191,-41.174,178.810,5.780,149.382
C01292=1168.960,-116.941,-41.183,178.812,5.781,149.381
C01293=1168.954,-116.691,-41.193,178.814,5.781,149.381
C01294=1168.948,-116.442,-41.201,178.816,5.781,149.380
C01295=1168.943,-116.192,-41.210,178.818,5.781,149.379
C01296=1168.938,-115.942,-41.219,178.821,5.782,149.379
C01297=1168.933,-115.692,-41.228,178.822,5.782,149.378
C01298=1168.928,-115.442,-41.237,178.824,5.783,149.378
C01299=1168.922,-115.192,-41.246,178.827,5.783,149.377
C01300=1168.917,-114.942,-41.255,178.829,5.783,149.377
C01301=1168.911,-114.693,-41.264,178.831,5.784,149.376
C01302=1168.906,-114.443,-41.273,178.833,5.783,149.375
C01303=1168.900,-114.193,-41.281,178.835,5.784,149.375
C01304=1168.895,-113.943,-41.290,178.837,5.784,149.374
C01305=1168.890,-113.694,-41.300,178.839,5.784,149.374
C01306=1168.885,-113.444,-41.309,178.841,5.784,149.373
C01307=1168.879,-113.194,-41.318,178.843,5.785,149.373
C01308=1168.874,-112.944,-41.327,178.845,5.785,149.372
C01309=1168.869,-112.695,-41.336,178.847,5.785,149.371
C01310=1168.863,-112.445,-41.345,178.849,5.785,149.371
C01311=1168.857,-112.195,-41.354,178.852,5.786,149.370
C01312=1168.852,-111.945,-41.363,178.853,5.786,149.370
C01313=1168.847,-111.696,-41.372,178.856,5.786,149.369
C01314=1168.842,-111.446,-41.382,178.858,5.786,149.369
C01315=1168.836,-111.196,-41.391,178.860,5.787,149.368
C01316=1168.831,-110.946,-41.400,178.862,5.787,149.367
C01317=1168.826,-110.696,-41.409,178.864,5.787,149.367
C01318=1168.821,-110.447,-41.418,178.866,5.788,149.366
C01319=1168.815,-110.196,-41.427,178.868,5.788,149.366
C01320=1168.810,-109.947,-41.437,178.871,5.788,149.365
C01321=1168.805,-109.697,-41.446,178.872,5.788,149.365
C01322=1168.800,-109.447,-41.455,178.875,5.789,149.364
C01323=1168.794,-109.197,-41.464,178.876,5.789,149.364
C01324=1168.789,-108.947,-41.473,178.879,5.789,149.363
C01325=1168.783,-108.699,-41.482,178.881,5.789,149.362
C01326=1168.778,-108.449,-41.491,178.883,5.790,149.362
C01327=1168.772,-108.199,-41.501,178.886,5.790,149.361
C01328=1168.767,-107.949,-41.510,178.887,5.790,149.361
C01329=1168.762,-107.700,-41.519,178.889,5.791,149.360
C01330=1168.756,-107.450,-41.529,178.891,5.791,149.359
C01331=1168.751,-107.200,-41.538,178.894,5.791,149.359
C01332=1168.746,-106.950,-41.547,178.896,5.791,149.358
C01333=1168.740,-106.700,-41.557,178.898,5.792,149.358
C01334=1168.735,-106.451,-41.566,178.899,5.792,149.357
C01335=1168.730,-106.201,-41.575,178.902,5.792,149.357
C01336=1168.725,-105.951,-41.583,178.904,5.793,149.356
C01337=1168.719,-105.701,-41.594,178.906,5.792,149.355
C01338=1168.714,-105.451,-41.603,178.909,5.793,149.355
C01339=1168.709,-105.202,-41.611,178.910,5.793,149.354
C01340=1168.703,-104.952,-41.622,178.913,5.793,149.354
C01341=1168.698,-104.702,-41.631,178.914,5.793,149.353
C01342=1168.692,-104.452,-41.640,178.917,5.794,149.352
C01343=1168.687,-104.203,-41.650,178.919,5.794,149.352
C01344=1168.682,-103.953,-41.659,178.921,5.795,149.352
C01345=1168.676,-103.703,-41.668,178.924,5.795,149.351
C01346=1168.671,-103.454,-41.678,178.925,5.795,149.350
C01347=1168.666,-103.204,-41.687,178.928,5.795,149.350
C01348=1168.660,-102.954,-41.696,178.929,5.795,149.349
C01349=1168.655,-102.704,-41.706,178.932,5.796,149.349
C01350=1168.650,-102.432,-41.716,178.934,5.796,149.348
C01351=1168.644,-102.160,-41.727,178.936,5.796,149.347
C01352=1168.638,-101.888,-41.737,178.939,5.797,149.347
C01353=1168.633,-101.616,-41.747,178.941,5.797,149.346
C01354=1168.628,-101.366,-41.756,178.943,5.797,149.346
C01355=1168.622,-101.117,-41.766,178.946,5.798,149.345
C01356=1168.617,-100.867,-41.775,178.947,5.798,149.344
C01357=1168.611,-100.617,-41.785,178.950,5.798,149.344
C01358=1168.606,-100.368,-41.794,178.952,5.799,149.343
C01359=1168.601,-100.118,-41.803,178.954,5.799,149.343
C01360=1168.595,-99.868,-41.813,178.956,5.799,149.342
C01361=1168.590,-99.618,-41.822,178.958,5.799,149.341
C01362=1168.584,-99.369,-41.832,178.961,5.799,149.341
C01363=1168.579,-99.119,-41.841,178.963,5.800,149.340
C01364=1168.574,-98.870,-41.852,178.964,5.800,149.340
C01365=1168.569,-98.620,-41.860,178.967,5.801,149.339
C01366=1168.564,-98.369,-41.871,178.969,5.801,149.339
C01367=1168.558,-98.120,-41.880,178.971,5.801,149.338
C01368=1168.553,-97.870,-41.890,178.973,5.801,149.337
C01369=1168.548,-97.620,-41.899,178.976,5.801,149.337
C01370=1168.542,-97.371,-41.909,178.978,5.802,149.336
C01371=1168.537,-97.121,-41.918,178.979,5.802,149.336
C01372=1168.531,-96.871,-41.928,178.982,5.802,149.335
C01373=1168.526,-96.621,-41.937,178.984,5.802,149.335
C01374=1168.520,-96.372,-41.947,178.986,5.803,149.334
C01375=1168.515,-96.122,-41.956,178.989,5.804,149.333
C01376=1168.510,-95.872,-41.967,178.991,5.803,149.333
C01377=1168.505,-95.622,-41.976,178.993,5.804,149.332
C01378=1168.500,-95.372,-41.986,178.994,5.804,149.332
C01379=1168.494,-95.122,-41.995,178.997,5.804,149.331
C01380=1168.489,-94.873,-42.005,178.999,5.805,149.330
C01381=1168.484,-94.624,-42.015,179.001,5.805,149.330
C01382=1168.478,-94.374,-42.024,179.004,5.805,149.329
C01383=1168.473,-94.123,-42.035,179.006,5.805,149.329
C01384=1168.468,-93.873,-42.044,179.008,5.806,149.328
C01385=1168.462,-93.624,-42.054,179.010,5.807,149.328
C01386=1168.457,-93.375,-42.064,179.012,5.806,149.327
C01387=1168.451,-93.125,-42.073,179.014,5.807,149.326
C01388=1168.447,-92.875,-42.083,179.016,5.807,149.326
C01389=1168.441,-92.626,-42.093,179.019,5.807,149.325
C01390=1168.436,-92.375,-42.103,179.021,5.808,149.324
C01391=1168.431,-92.126,-42.112,179.023,5.808,149.324
C01392=1168.425,-91.876,-42.123,179.026,5.808,149.323
C01393=1168.420,-91.626,-42.131,179.028,5.809,149.323
C01394=1168.414,-91.377,-42.142,179.029,5.809,149.322
C01395=1168.409,-91.126,-42.152,179.032,5.809,149.322
C01396=1168.404,-90.877,-42.161,179.034,5.809,149.321
C01397=1168.399,-90.627,-42.171,179.036,5.810,149.320
C01398=1168.393,-90.378,-42.182,179.038,5.810,149.320
C01399=1168.388,-90.128,-42.190,179.041,5.810,149.319
C01400=1168.383,-89.877,-42.201,179.043,5.811,149.319
C01401=1168.378,-89.628,-42.211,179.045,5.810,149.318
C01402=1168.373,-89.379,-42.221,179.047,5.811,149.318
C01403=1168.367,-89.128,-42.230,179.050,5.811,149.317
C01404=1168.362,-88.879,-42.240,179.051,5.811,149.316
C01405=1168.357,-88.629,-42.251,179.054,5.812,149.316
C01406=1168.351,-88.379,-42.261,179.056,5.813,149.315
C01407=1168.346,-88.130,-42.270,179.058,5.813,149.315
C01408=1168.340,-87.880,-42.280,179.060,5.813,149.314
C01409=1168.335,-87.630,-42.290,179.062,5.813,149.313
C01410=1168.331,-87.381,-42.300,179.065,5.813,149.313
C01411=1168.325,-87.130,-42.310,179.067,5.814,149.312
C01412=1168.319,-86.881,-42.320,179.069,5.814,149.312
C01413=1168.313,-86.631,-42.330,179.071,5.815,149.311
C01414=1168.309,-86.381,-42.340,179.074,5.815,149.310
C01415=1168.304,-86.132,-42.350,179.075,5.815,149.310
C01416=1168.298,-85.882,-42.360,179.078,5.815,149.309
C01417=1168.293,-85.632,-42.370,179.080,5.816,149.309
C01418=1168.288,-85.382,-42.380,179.082,5.816,149.308
C01419=1168.282,-85.133,-42.390,179.085,5.816,149.307
C01420=1168.277,-84.883,-42.400,179.087,5.816,149.307
C01421=1168.272,-84.633,-42.410,179.089,5.817,149.306
C01422=1168.267,-84.384,-42.420,179.091,5.818,149.306
C01423=1168.261,-84.134,-42.430,179.093,5.817,149.305
C01424=1168.256,-83.884,-42.440,179.095,5.818,149.305
C01425=1168.251,-83.634,-42.450,179.098,5.818,149.304
C01426=1168.245,-83.384,-42.460,179.099,5.818,149.303
C01427=1168.240,-83.135,-42.471,179.102,5.819,149.303
C01428=1168.235,-82.885,-42.481,179.104,5.820,149.302
C01429=1168.230,-82.635,-42.491,179.106,5.819,149.302
C01430=1168.224,-82.386,-42.501,179.109,5.820,149.301
C01431=1168.219,-82.136,-42.511,179.111,5.820,149.300
C01432=1168.214,-81.886,-42.522,179.113,5.820,149.300
C01433=1168.208,-81.637,-42.532,179.116,5.821,149.299
C01434=1168.204,-81.387,-42.542,179.118,5.821,149.299
C01435=1168.198,-81.137,-42.552,179.120,5.821,149.298
C01436=1168.192,-80.887,-42.562,179.122,5.822,149.297
C01437=1168.187,-80.637,-42.572,179.125,5.822,149.297
C01438=1168.182,-80.387,-42.582,179.126,5.822,149.296
C01439=1168.177,-80.138,-42.592,179.129,5.823,149.296
C01440=1168.171,-79.888,-42.602,179.131,5.823,149.295
C01441=1168.166,-79.638,-42.613,179.133,5.823,149.294
C01442=1168.161,-79.389,-42.623,179.135,5.824,149.294
C01443=1168.156,-79.138,-42.634,179.137,5.823,149.293
C01444=1168.150,-78.889,-42.644,179.140,5.824,149.293
C01445=1168.145,-78.639,-42.654,179.142,5.825,149.292
C01446=1168.140,-78.389,-42.664,179.144,5.825,149.292
C01447=1168.135,-78.140,-42.675,179.147,5.825,149.291
C01448=1168.129,-77.891,-42.685,179.149,5.826,149.290
C01449=1168.124,-77.641,-42.696,179.151,5.826,149.290
C01450=1168.119,-77.391,-42.706,179.153,5.826,149.289
C01451=1168.113,-77.142,-42.716,179.156,5.827,149.288
C01452=1168.108,-76.891,-42.727,179.158,5.827,149.288
C01453=1168.103,-76.642,-42.737,179.160,5.827,149.287
C01454=1168.097,-76.370,-42.748,179.162,5.828,149.287
C01455=1168.091,-76.100,-42.759,179.165,5.828,149.286
C01456=1168.086,-75.828,-42.770,179.168,5.828,149.285
C01457=1168.080,-75.557,-42.782,179.169,5.828,149.285
C01458=1168.074,-75.308,-42.792,179.172,5.829,149.284
C01459=1168.069,-75.057,-42.803,179.174,5.830,149.284
C01460=1168.064,-74.808,-42.813,179.177,5.830,149.283
C01461=1168.058,-74.558,-42.823,179.178,5.830,149.282
C01462=1168.053,-74.308,-42.834,179.181,5.830,149.282
C01463=1168.048,-74.059,-42.844,179.183,5.831,149.281
C01464=1168.043,-73.809,-42.855,179.185,5.831,149.281
C01465=1168.037,-73.559,-42.866,179.188,5.831,149.280
C01466=1168.032,-73.310,-42.876,179.190,5.832,149.279
C01467=1168.027,-73.060,-42.886,179.192,5.832,149.279
C01468=1168.021,-72.810,-42.897,179.194,5.832,149.278
C01469=1168.016,-72.560,-42.907,179.197,5.833,149.277
C01470=1168.011,-72.311,-42.918,179.199,5.833,149.277
C01471=1168.006,-72.061,-42.929,179.201,5.833,149.276
C01472=1168.000,-71.811,-42.939,179.203,5.834,149.276
C01473=1167.995,-71.562,-42.949,179.206,5.834,149.275
C01474=1167.990,-71.312,-42.960,179.208,5.834,149.275
C01475=1167.984,-71.062,-42.971,179.210,5.835,149.274
C01476=1167.979,-70.812,-42.981,179.213,5.836,149.273
C01477=1167.974,-70.563,-42.991,179.215,5.835,149.273
C01478=1167.969,-70.313,-43.003,179.217,5.836,149.272
C01479=1167.964,-70.063,-43.013,179.220,5.836,149.272
C01480=1167.959,-69.813,-43.023,179.221,5.836,149.271
C01481=1167.953,-69.564,-43.034,179.224,5.837,149.270
C01482=1167.948,-69.314,-43.045,179.226,5.838,149.270
C01483=1167.943,-69.065,-43.055,179.229,5.838,149.269
C01484=1167.938,-68.814,-43.066,179.230,5.838,149.269
C01485=1167.932,-68.565,-43.077,179.233,5.838,149.268
C01486=1167.927,-68.315,-43.087,179.235,5.839,149.268
C01487=1167.922,-68.066,-43.097,179.237,5.839,149.267
C01488=1167.917,-67.816,-43.109,179.239,5.840,149.266
C01489=1167.911,-67.566,-43.119,179.242,5.840,149.266
C01490=1167.906,-67.316,-43.130,179.244,5.841,149.265
C01491=1167.900,-67.067,-43.141,179.246,5.840,149.264
C01492=1167.895,-66.817,-43.152,179.248,5.841,149.264
C01493=1167.890,-66.567,-43.162,179.251,5.842,149.263
C01494=1167.885,-66.318,-43.173,179.253,5.841,149.263
C01495=1167.880,-66.068,-43.183,179.255,5.842,149.262
C01496=1167.875,-65.818,-43.194,179.258,5.842,149.261
C01497=1167.869,-65.569,-43.205,179.260,5.843,149.261
C01498=1167.864,-65.319,-43.215,179.262,5.843,149.260
C01499=1167.858,-65.069,-43.227,179.265,5.844,149.260
C01500=1167.853,-64.819,-43.237,179.267,5.844,149.259
C01501=1167.848,-64.570,-43.248,179.269,5.844,149.259
C01502=1167.843,-64.320,-43.259,179.271,5.844,149.258
C01503=1167.838,-64.070,-43.270,179.274,5.845,149.257
C01504=1167.833,-63.821,-43.280,179.276,5.846,149.257
C01505=1167.827,-63.570,-43.292,179.278,5.846,149.256
C01506=1167.822,-63.321,-43.303,179.281,5.846,149.255
C01507=1167.817,-63.071,-43.313,179.283,5.847,149.255
C01508=1167.811,-62.822,-43.324,179.285,5.847,149.254
C01509=1167.806,-62.572,-43.335,179.288,5.847,149.254
C01510=1167.802,-62.322,-43.346,179.290,5.848,149.253
C01511=1167.795,-62.072,-43.357,179.292,5.848,149.252
C01512=1167.791,-61.823,-43.368,179.295,5.849,149.252
C01513=1167.785,-61.573,-43.378,179.297,5.848,149.251
C01514=1167.780,-61.324,-43.390,179.299,5.849,149.251
C01515=1167.775,-61.073,-43.401,179.302,5.850,149.250
C01516=1167.769,-60.824,-43.412,179.304,5.850,149.250
C01517=1167.764,-60.574,-43.422,179.306,5.850,149.249
C01518=1167.759,-60.325,-43.433,179.308,5.851,149.248
C01519=1167.754,-60.075,-43.444,179.311,5.851,149.248
C01520=1167.749,-59.825,-43.456,179.313,5.852,149.247
C01521=1167.743,-59.576,-43.467,179.315,5.852,149.246
C01522=1167.738,-59.326,-43.477,179.318,5.852,149.246
C01523=1167.734,-59.076,-43.488,179.320,5.853,149.245
C01524=1167.727,-58.826,-43.499,179.322,5.853,149.245
C01525=1167.723,-58.576,-43.510,179.324,5.853,149.244
C01526=1167.717,-58.328,-43.521,179.327,5.854,149.243
C01527=1167.712,-58.077,-43.533,179.329,5.854,149.243
C01528=1167.707,-57.827,-43.544,179.332,5.855,149.242
C01529=1167.701,-57.578,-43.554,179.333,5.855,149.242
C01530=1167.697,-57.328,-43.565,179.336,5.855,149.241
C01531=1167.691,-57.078,-43.577,179.338,5.856,149.240
C01532=1167.686,-56.829,-43.587,179.341,5.856,149.240
C01533=1167.681,-56.579,-43.599,179.343,5.856,149.239
C01534=1167.675,-56.329,-43.611,179.345,5.857,149.239
C01535=1167.670,-56.080,-43.621,179.348,5.857,149.238
C01536=1167.665,-55.830,-43.632,179.350,5.858,149.237
C01537=1167.660,-55.580,-43.644,179.352,5.858,149.237
C01538=1167.654,-55.331,-43.654,179.354,5.858,149.236
C01539=1167.649,-55.081,-43.666,179.357,5.859,149.236
C01540=1167.644,-54.831,-43.677,179.359,5.859,149.235
C01541=1167.639,-54.581,-43.689,179.362,5.860,149.234
C01542=1167.634,-54.332,-43.699,179.364,5.860,149.234
C01543=1167.628,-54.082,-43.711,179.366,5.860,149.233
C01544=1167.624,-53.832,-43.722,179.368,5.861,149.232
C01545=1167.618,-53.583,-43.733,179.371,5.862,149.232
C01546=1167.613,-53.333,-43.744,179.373,5.861,149.231
C01547=1167.608,-53.083,-43.755,179.375,5.862,149.231
C01548=1167.602,-52.833,-43.767,179.378,5.863,149.230
C01549=1167.597,-52.584,-43.778,179.380,5.863,149.229
C01550=1167.592,-52.334,-43.789,179.382,5.864,149.229
C01551=1167.587,-52.084,-43.801,179.384,5.863,149.228
C01552=1167.581,-51.835,-43.812,179.387,5.864,149.228
C01553=1167.576,-51.585,-43.824,179.389,5.865,149.227
C01554=1167.571,-51.336,-43.835,179.392,5.865,149.227
C01555=1167.566,-51.085,-43.846,179.394,5.866,149.226
C01556=1167.560,-50.836,-43.857,179.396,5.866,149.225
C01557=1167.556,-50.586,-43.868,179.398,5.866,149.225
C01558=1167.550,-50.316,-43.881,179.401,5.867,149.224
C01559=1167.544,-50.046,-43.893,179.404,5.867,149.223
C01560=1167.538,-49.775,-43.905,179.406,5.868,149.223
C01561=1167.533,-49.505,-43.918,179.409,5.868,149.222
C01562=1167.528,-49.256,-43.929,179.411,5.869,149.221
C01563=1167.522,-49.005,-43.940,179.413,5.869,149.221
C01564=1167.517,-48.755,-43.952,179.416,5.869,149.220
C01565=1167.512,-48.505,-43.964,179.418,5.870,149.220
C01566=1167.507,-48.257,-43.974,179.420,5.870,149.219
C01567=1167.501,-48.007,-43.986,179.423,5.871,149.218
C01568=1167.497,-47.757,-43.998,179.425,5.872,149.218
C01569=1167.491,-47.507,-44.010,179.427,5.871,149.217
C01570=1167.486,-47.257,-44.021,179.430,5.872,149.217
C01571=1167.480,-47.008,-44.032,179.432,5.872,149.216
C01572=1167.475,-46.758,-44.044,179.434,5.873,149.216
C01573=1167.470,-46.509,-44.056,179.437,5.874,149.215
C01574=1167.465,-46.259,-44.067,179.439,5.874,149.214
C01575=1167.460,-46.009,-44.079,179.441,5.874,149.214
C01576=1167.454,-45.760,-44.090,179.444,5.874,149.213
C01577=1167.449,-45.510,-44.101,179.446,5.875,149.212
C01578=1167.444,-45.260,-44.113,179.449,5.876,149.212
C01579=1167.439,-45.011,-44.125,179.451,5.876,149.211
C01580=1167.434,-44.761,-44.137,179.453,5.876,149.211
C01581=1167.428,-44.511,-44.148,179.455,5.877,149.210
C01582=1167.423,-44.262,-44.159,179.458,5.877,149.209
C01583=1167.418,-44.012,-44.171,179.461,5.878,149.209
C01584=1167.413,-43.762,-44.183,179.463,5.879,149.208
C01585=1167.408,-43.512,-44.194,179.465,5.878,149.208
C01586=1167.402,-43.262,-44.206,179.467,5.879,149.207
C01587=1167.398,-43.013,-44.218,179.470,5.879,149.206
C01588=1167.392,-42.763,-44.229,179.472,5.880,149.206
C01589=1167.387,-42.514,-44.240,179.475,5.881,149.205
C01590=1167.381,-42.264,-44.252,179.477,5.881,149.204
C01591=1167.376,-42.014,-44.264,179.479,5.881,149.204
C01592=1167.371,-41.764,-44.275,179.481,5.881,149.203
C01593=1167.366,-41.514,-44.287,179.484,5.882,149.203
C01594=1167.361,-41.265,-44.300,179.486,5.883,149.202
C01595=1167.356,-41.016,-44.311,179.489,5.883,149.201
C01596=1167.351,-40.766,-44.323,179.491,5.884,149.201
C01597=1167.345,-40.517,-44.334,179.493,5.884,149.200
C01598=1167.340,-40.267,-44.346,179.495,5.884,149.200
C01599=1167.334,-40.017,-44.358,179.498,5.885,149.199
C01600=1167.329,-39.767,-44.370,179.500,5.886,149.199
C01601=1167.325,-39.518,-44.382,179.503,5.886,149.198
C01602=1167.319,-39.268,-44.394,179.506,5.886,149.197
C01603=1167.314,-39.018,-44.405,179.508,5.887,149.197
C01604=1167.309,-38.768,-44.417,179.510,5.887,149.196
C01605=1167.304,-38.518,-44.429,179.512,5.888,149.196
C01606=1167.298,-38.269,-44.441,179.515,5.888,149.195
C01607=1167.293,-38.019,-44.453,179.517,5.889,149.194
C01608=1167.288,-37.770,-44.464,179.520,5.889,149.194
C01609=1167.282,-37.520,-44.476,179.522,5.890,149.193
C01610=1167.277,-37.270,-44.488,179.524,5.891,149.193
C01611=1167.273,-37.021,-44.500,179.526,5.890,149.192
C01612=1167.267,-36.771,-44.512,179.529,5.891,149.191
C01613=1167.262,-36.521,-44.524,179.531,5.891,149.191
C01614=1167.257,-36.272,-44.536,179.534,5.892,149.190
C01615=1167.252,-36.023,-44.548,179.536,5.893,149.189
C01616=1167.246,-35.773,-44.559,179.539,5.893,149.189
C01617=1167.241,-35.523,-44.571,179.541,5.894,149.188
C01618=1167.236,-35.273,-44.584,179.543,5.893,149.188
C01619=1167.230,-35.023,-44.596,179.545,5.894,149.187
C01620=1167.226,-34.774,-44.607,179.548,5.895,149.186
C01621=1167.221,-34.524,-44.620,179.551,5.895,149.186
C01622=1167.215,-34.275,-44.632,179.553,5.896,149.185
C01623=1167.210,-34.025,-44.643,179.555,5.896,149.185
C01624=1167.205,-33.775,-44.656,179.558,5.897,149.184
C01625=1167.200,-33.526,-44.667,179.560,5.898,149.183
C01626=1167.195,-33.276,-44.679,179.562,5.897,149.183
C01627=1167.189,-33.026,-44.692,179.564,5.898,149.182
C01628=1167.184,-32.776,-44.704,179.567,5.898,149.182
C01629=1167.179,-32.527,-44.716,179.569,5.899,149.181
C01630=1167.173,-32.277,-44.728,179.572,5.900,149.180
C01631=1167.169,-32.028,-44.739,179.574,5.901,149.180
C01632=1167.164,-31.778,-44.752,179.577,5.901,149.179
C01633=1167.158,-31.528,-44.764,179.580,5.901,149.178
C01634=1167.153,-31.279,-44.777,179.582,5.902,149.178
C01635=1167.148,-31.029,-44.788,179.584,5.902,149.177
C01636=1167.142,-30.779,-44.800,179.586,5.903,149.177
C01637=1167.137,-30.530,-44.813,179.589,5.903,149.176
C01638=1167.132,-30.280,-44.825,179.591,5.904,149.175
C01639=1167.127,-30.031,-44.837,179.593,5.904,149.175
C01640=1167.122,-29.781,-44.849,179.596,5.905,149.174
C01641=1167.117,-29.532,-44.861,179.598,5.906,149.174
C01642=1167.111,-29.282,-44.873,179.601,5.906,149.173
C01643=1167.106,-29.032,-44.886,179.604,5.906,149.172
C01644=1167.101,-28.782,-44.898,179.606,5.907,149.172
C01645=1167.096,-28.532,-44.911,179.608,5.907,149.171
C01646=1167.091,-28.282,-44.923,179.610,5.908,149.171
C01647=1167.086,-28.033,-44.935,179.613,5.908,149.170
C01648=1167.080,-27.783,-44.947,179.615,5.909,149.170
C01649=1167.075,-27.534,-44.960,179.618,5.909,149.169
C01650=1167.070,-27.285,-44.972,179.620,5.910,149.168
C01651=1167.065,-27.035,-44.984,179.622,5.911,149.168
C01652=1167.059,-26.785,-44.997,179.625,5.911,149.167
C01653=1167.054,-26.535,-45.009,179.627,5.912,149.167
C01654=1167.050,-26.286,-45.021,179.630,5.912,149.166
C01655=1167.045,-26.036,-45.033,179.633,5.913,149.165
C01656=1167.040,-25.786,-45.045,179.634,5.913,149.165
C01657=1167.035,-25.537,-45.058,179.637,5.913,149.164
C01658=1167.029,-25.287,-45.070,179.639,5.914,149.164
C01659=1167.024,-25.038,-45.083,179.642,5.914,149.163
C01660=1167.019,-24.788,-45.094,179.644,5.915,149.162
C01661=1167.013,-24.539,-45.107,179.646,5.916,149.162
C01662=1167.008,-24.269,-45.121,179.649,5.916,149.161
C01663=1167.002,-23.998,-45.134,179.652,5.917,149.160
C01664=1166.997,-23.729,-45.148,179.654,5.917,149.160
C01665=1166.991,-23.459,-45.161,179.657,5.918,149.159
C01666=1166.986,-23.209,-45.174,179.659,5.918,149.158
C01667=1166.980,-22.960,-45.186,179.662,5.919,149.158
C01668=1166.975,-22.710,-45.198,179.664,5.919,149.157
C01669=1166.970,-22.460,-45.211,179.667,5.920,149.157
C01670=1166.965,-22.211,-45.224,179.669,5.921,149.156
C01671=1166.960,-21.961,-45.236,179.672,5.921,149.155
C01672=1166.955,-21.711,-45.248,179.674,5.922,149.155
C01673=1166.950,-21.462,-45.261,179.676,5.922,149.154
C01674=1166.945,-21.213,-45.273,179.679,5.923,149.154
C01675=1166.939,-20.962,-45.287,179.681,5.924,149.153
C01676=1166.934,-20.712,-45.299,179.684,5.924,149.152
C01677=1166.929,-20.463,-45.312,179.686,5.925,149.152
C01678=1166.924,-20.214,-45.324,179.689,5.925,149.151
C01679=1166.919,-19.965,-45.337,179.691,5.926,149.150
C01680=1166.914,-19.714,-45.349,179.693,5.926,149.150
C01681=1166.909,-19.465,-45.362,179.696,5.926,149.149
C01682=1166.903,-19.215,-45.374,179.698,5.927,149.149
C01683=1166.898,-18.966,-45.387,179.701,5.928,149.148
C01684=1166.892,-18.716,-45.400,179.703,5.928,149.147
C01685=1166.888,-18.466,-45.413,179.705,5.929,149.147
C01686=1166.882,-18.216,-45.425,179.708,5.929,149.146
C01687=1166.877,-17.967,-45.437,179.710,5.930,149.146
C01688=1166.872,-17.718,-45.450,179.713,5.930,149.145
C01689=1166.867,-17.467,-45.464,179.716,5.931,149.144
C01690=1166.862,-17.218,-45.476,179.718,5.932,149.144
C01691=1166.857,-16.969,-45.489,179.720,5.932,149.143
C01692=1166.852,-16.719,-45.501,179.723,5.933,149.143
C01693=1166.846,-16.469,-45.513,179.725,5.933,149.142
C01694=1166.841,-16.219,-45.527,179.728,5.934,149.141
C01695=1166.836,-15.970,-45.539,179.730,5.935,149.141
C01696=1166.831,-15.721,-45.552,179.733,5.935,149.140
C01697=1166.826,-15.470,-45.565,179.735,5.936,149.140
C01698=1166.821,-15.221,-45.578,179.738,5.936,149.139
C01699=1166.815,-14.972,-45.591,179.740,5.937,149.138
C01700=1166.810,-14.722,-45.603,179.742,5.938,149.138
C01701=1166.806,-14.472,-45.616,179.745,5.938,149.137
C01702=1166.800,-14.223,-45.629,179.747,5.939,149.137
C01703=1166.795,-13.973,-45.642,179.750,5.939,149.136
C01704=1166.790,-13.723,-45.655,179.753,5.940,149.135
C01705=1166.785,-13.474,-45.668,179.755,5.941,149.135
C01706=1166.780,-13.225,-45.680,179.757,5.941,149.134
C01707=1166.774,-12.975,-45.694,179.760,5.942,149.134
C01708=1166.769,-12.725,-45.706,179.762,5.942,149.133
C01709=1166.764,-12.476,-45.719,179.765,5.943,149.132
C01710=1166.758,-12.226,-45.732,179.767,5.944,149.132
C01711=1166.754,-11.976,-45.745,179.770,5.944,149.131
C01712=1166.749,-11.727,-45.758,179.772,5.945,149.131
C01713=1166.743,-11.477,-45.771,179.775,5.945,149.130
C01714=1166.738,-11.227,-45.784,179.777,5.946,149.130
C01715=1166.733,-10.978,-45.797,179.779,5.947,149.129
C01716=1166.727,-10.728,-45.810,179.782,5.947,149.128
C01717=1166.723,-10.478,-45.823,179.784,5.948,149.128
C01718=1166.718,-10.229,-45.836,179.787,5.948,149.127
C01719=1166.713,-9.979,-45.850,179.789,5.949,149.127
C01720=1166.708,-9.730,-45.862,179.792,5.950,149.126
C01721=1166.703,-9.480,-45.875,179.794,5.950,149.125
C01722=1166.697,-9.230,-45.888,179.797,5.951,149.125
C01723=1166.692,-8.981,-45.901,179.799,5.951,149.124
C01724=1166.687,-8.731,-45.914,179.801,5.952,149.124
C01725=1166.682,-8.482,-45.928,179.804,5.953,149.123
C01726=1166.677,-8.232,-45.940,179.807,5.953,149.122
C01727=1166.672,-7.982,-45.953,179.809,5.954,149.122
C01728=1166.667,-7.733,-45.967,179.812,5.954,149.121
C01729=1166.661,-7.483,-45.979,179.814,5.955,149.121
C01730=1166.656,-7.233,-45.993,179.816,5.956,149.120
C01731=1166.651,-6.984,-46.006,179.819,5.956,149.119
C01732=1166.646,-6.734,-46.020,179.821,5.957,149.119
C01733=1166.641,-6.485,-46.032,179.824,5.957,149.118
C01734=1166.636,-6.235,-46.045,179.826,5.958,149.118
C01735=1166.631,-5.986,-46.059,179.829,5.959,149.117
C01736=1166.626,-5.736,-46.072,179.831,5.959,149.116
C01737=1166.621,-5.486,-46.085,179.833,5.960,149.116
C01738=1166.615,-5.237,-46.098,179.836,5.960,149.115
C01739=1166.610,-4.988,-46.112,179.838,5.961,149.115
C01740=1166.605,-4.738,-46.125,179.841,5.962,149.114
C01741=1166.599,-4.488,-46.138,179.844,5.962,149.113
C01742=1166.595,-4.238,-46.151,179.846,5.963,149.113
C01743=1166.589,-3.989,-46.165,179.848,5.963,149.112
C01744=1166.585,-3.739,-46.178,179.851,5.964,149.112
C01745=1166.579,-3.489,-46.191,179.853,5.965,149.111
C01746=1166.575,-3.240,-46.205,179.855,5.965,149.110
C01747=1166.569,-2.990,-46.218,179.858,5.966,149.110
C01748=1166.564,-2.740,-46.231,179.861,5.966,149.109
C01749=1166.559,-2.491,-46.245,179.863,5.967,149.109
C01750=1166.554,-2.242,-46.257,179.866,5.968,149.108
C01751=1166.549,-1.992,-46.272,179.868,5.968,149.107
C01752=1166.544,-1.743,-46.284,179.870,5.969,149.107
C01753=1166.538,-1.493,-46.298,179.873,5.969,149.106
C01754=1166.534,-1.244,-46.311,179.876,5.971,149.106
C01755=1166.528,-0.994,-46.325,179.878,5.971,149.105
C01756=1166.522,-0.744,-46.338,179.881,5.972,149.104
C01757=1166.518,-0.495,-46.352,179.883,5.973,149.104
C01758=1166.512,-0.245,-46.365,179.886,5.973,149.103
C01759=1166.508,0.004,-46.378,179.888,5.974,149.103
C01760=1166.502,0.254,-46.392,179.891,5.974,149.102
C01761=1166.498,0.503,-46.405,179.893,5.975,149.101
C01762=1166.492,0.753,-46.419,179.896,5.976,149.101
C01763=1166.487,1.003,-46.433,179.898,5.977,149.100
C01764=1166.483,1.253,-46.446,179.900,5.977,149.100
C01765=1166.477,1.502,-46.460,179.903,5.977,149.099
C01766=1166.471,1.772,-46.474,179.905,5.978,149.098
C01767=1166.466,2.041,-46.489,179.909,5.980,149.098
C01768=1166.461,2.310,-46.503,179.911,5.980,149.097
C01769=1166.455,2.579,-46.518,179.914,5.980,149.096
C01770=1166.450,2.829,-46.532,179.916,5.981,149.096
C01771=1166.445,3.078,-46.545,179.919,5.982,149.095
C01772=1166.440,3.328,-46.558,179.921,5.982,149.095
C01773=1166.434,3.577,-46.572,179.923,5.983,149.094
C01774=1166.430,3.827,-46.585,179.927,5.984,149.093
C01775=1166.424,4.076,-46.599,179.929,5.985,149.093
C01776=1166.419,4.326,-46.614,179.932,5.986,149.092
C01777=1166.414,4.576,-46.627,179.934,5.986,149.092
C01778=1166.409,4.825,-46.640,179.936,5.987,149.091
C01779=1166.404,5.075,-46.654,179.939,5.987,149.090
C01780=1166.398,5.324,-46.668,179.941,5.988,149.090
C01781=1166.394,5.574,-46.682,179.944,5.989,149.089
C01782=1166.389,5.824,-46.695,179.946,5.990,149.089
C01783=1166.383,6.073,-46.709,179.949,5.990,149.088
C01784=1166.378,6.323,-46.723,179.951,5.990,149.087
C01785=1166.373,6.572,-46.736,179.954,5.991,149.087
C01786=1166.368,6.822,-46.750,179.957,5.993,149.086
C01787=1166.363,7.072,-46.764,179.959,5.993,149.086
C01788=1166.358,7.321,-46.778,179.962,5.994,149.085
C01789=1166.353,7.571,-46.791,179.964,5.994,149.084
C01790=1166.348,7.820,-46.806,179.966,5.995,149.084
C01791=1166.343,8.070,-46.819,179.969,5.996,149.083
C01792=1166.338,8.320,-46.833,179.971,5.996,149.083
C01793=1166.333,8.568,-46.846,179.974,5.997,149.082
C01794=1166.328,8.818,-46.861,179.976,5.998,149.082
C01795=1166.323,9.069,-46.874,179.979,5.999,149.081
C01796=1166.317,9.318,-46.888,179.982,5.999,149.080
C01797=1166.312,9.567,-46.902,179.984,6.000,149.080
C01798=1166.308,9.817,-46.916,179.987,6.001,149.079
C01799=1166.302,10.066,-46.929,179.989,6.002,149.079
C01800=1166.297,10.316,-46.944,179.992,6.002,149.078
C01801=1166.292,10.566,-46.958,179.994,6.002,149.077
C01802=1166.286,10.815,-46.972,179.996,6.003,149.077
C01803=1166.282,11.064,-46.986,179.999,6.004,149.076
C01804=1166.277,11.314,-46.999,-179.998,6.005,149.076
C01805=1166.272,11.564,-47.013,-179.996,6.006,149.075
C01806=1166.266,11.813,-47.027,-179.993,6.007,149.075
C01807=1166.262,12.063,-47.041,-179.991,6.007,149.074
C01808=1166.257,12.313,-47.056,-179.988,6.008,149.073
C01809=1166.251,12.562,-47.070,-179.986,6.008,149.073
C01810=1166.246,12.811,-47.084,-179.983,6.009,149.072
C01811=1166.241,13.062,-47.097,-179.981,6.010,149.072
C01812=1166.235,13.311,-47.111,-179.978,6.011,149.071
C01813=1166.231,13.560,-47.125,-179.976,6.012,149.071
C01814=1166.226,13.810,-47.139,-179.973,6.012,149.070
C01815=1166.221,14.059,-47.154,-179.970,6.013,149.069
C01816=1166.216,14.308,-47.168,-179.968,6.014,149.069
C01817=1166.211,14.558,-47.182,-179.966,6.014,149.068
C01818=1166.206,14.808,-47.196,-179.963,6.015,149.068
C01819=1166.201,15.058,-47.210,-179.960,6.016,149.067
C01820=1166.195,15.307,-47.224,-179.957,6.017,149.066
C01821=1166.190,15.556,-47.239,-179.955,6.018,149.066
C01822=1166.185,15.806,-47.253,-179.953,6.018,149.065
C01823=1166.180,16.056,-47.267,-179.951,6.019,149.065
C01824=1166.175,16.305,-47.281,-179.948,6.019,149.064
C01825=1166.170,16.554,-47.295,-179.945,6.021,149.063
C01826=1166.165,16.804,-47.310,-179.942,6.021,149.063
C01827=1166.160,17.054,-47.324,-179.940,6.022,149.062
C01828=1166.155,17.304,-47.338,-179.938,6.023,149.062
C01829=1166.149,17.553,-47.352,-179.935,6.023,149.061
C01830=1166.144,17.802,-47.366,-179.933,6.024,149.061
C01831=1166.139,18.052,-47.381,-179.930,6.025,149.060
C01832=1166.134,18.302,-47.395,-179.927,6.026,149.059
C01833=1166.130,18.551,-47.409,-179.925,6.027,149.059
C01834=1166.124,18.800,-47.423,-179.922,6.027,149.058
C01835=1166.119,19.050,-47.437,-179.920,6.028,149.058
C01836=1166.114,19.300,-47.452,-179.917,6.028,149.057
C01837=1166.109,19.550,-47.466,-179.915,6.029,149.056
